DATA_BLOCK "BOTONERA"   // DB2
{ S7_Optimized_Access := 'TRUE' }
VERSION : 0.1
   VAR
      "096P005A" : Struct
         START : Bool;
         STOP : Bool;
         FALLA : Bool;
         "RESET FALLA" : Bool;
         "RESET TIEMPO OPERANDO" : Bool;
         "RESET TIEMPO ACUMULADO" : Bool;
      END_STRUCT;
      "096P005B" : Struct
         START : Bool;
         STOP : Bool;
         FALLA : Bool;
         "RESET FALLA" : Bool;
         "RESET TIEMPO OPERANDO" : Bool;
         "RESET TIEMPO ACUMULADO" : Bool;
      END_STRUCT;
      "096P004A" : Struct
         START : Bool;
         STOP : Bool;
         FALLA : Bool;
         "RESET FALLA" : Bool;
         "RESET TIEMPO OPERANDO" : Bool;
         "RESET TIEMPO ACUMULADO" : Bool;
      END_STRUCT;
      "096P004B" : Struct
         START : Bool;
         STOP : Bool;
         FALLA : Bool;
         "RESET FALLA" : Bool;
         "RESET TIEMPO OPERANDO" : Bool;
         "RESET TIEMPO ACUMULADO" : Bool;
      END_STRUCT;
      "096P004C" : Struct
         START : Bool;
         STOP : Bool;
         FALLA : Bool;
         "RESET FALLA" : Bool;
         "RESET TIEMPO OPERANDO" : Bool;
         "RESET TIEMPO ACUMULADO" : Bool;
      END_STRUCT;
      "096P004D" : Struct
         START : Bool;
         STOP : Bool;
         FALLA : Bool;
         "RESET FALLA" : Bool;
         "RESET TIEMPO OPERANDO" : Bool;
         "RESET TIEMPO ACUMULADO" : Bool;
      END_STRUCT;
      "TODO A MANUAL" : Bool;
      "TODO A AUTOMATICO" : Bool;
      "TODO EN MANUAL" : Bool;
      "TODO EN AUTOMATICO" : Bool;
   END_VAR
BEGIN
END_DATA_BLOCK

DATA_BLOCK "MODO OPERACION"   // DB3
{ S7_Optimized_Access := 'TRUE' }
VERSION : 0.1
   VAR RETAIN
      "096P004A" : Struct
         MANUAL : Bool;
         AUTOMATICO : Bool;
         SCADA : Bool;
      END_STRUCT;
      "096P004B" : Struct
         MANUAL : Bool;
         AUTOMATICO : Bool;
         SCADA : Bool;
      END_STRUCT;
      "096P004C" : Struct
         MANUAL : Bool;
         AUTOMATICO : Bool;
         SCADA : Bool;
      END_STRUCT;
      "096P004D" : Struct
         MANUAL : Bool;
         AUTOMATICO : Bool;
         SCADA : Bool;
      END_STRUCT;
      "096P005A" : Struct
         MANUAL : Bool;
         AUTOMATICO : Bool;
         SCADA : Bool;
      END_STRUCT;
      "096P005B" : Struct
         MANUAL : Bool;
         AUTOMATICO : Bool;
         SCADA : Bool;
      END_STRUCT;
   END_VAR
BEGIN
END_DATA_BLOCK

DATA_BLOCK "ESC HZ"   // DB4
{ S7_Optimized_Access := 'TRUE' }
VERSION : 0.1
   VAR RETAIN
      "096P004A" : Struct
         "FRECUENCIA MAX" : Real := 60.0;
         "FRECUENCIA MIN" : Real := 20.0;
         "FRECUENCIA OP" : Real := 60.0;
      END_STRUCT;
      "096P004B" : Struct
         "FRECUENCIA MAX" : Real := 60.0;
         "FRECUENCIA MIN" : Real := 20.0;
         "FRECUENCIA OP" : Real := 60.0;
      END_STRUCT;
      "096P004C" : Struct
         "FRECUENCIA MAX" : Real := 60.0;
         "FRECUENCIA MIN" : Real := 20.0;
         "FRECUENCIA OP" : Real := 60.0;
      END_STRUCT;
      "096P004D" : Struct
         "FRECUENCIA MAX" : Real := 60.0;
         "FRECUENCIA MIN" : Real := 20.0;
         "FRECUENCIA OP" : Real := 60.0;
      END_STRUCT;
   END_VAR
BEGIN
END_DATA_BLOCK

DATA_BLOCK "DATOS LECTURA VFDS"   // DB5
{ S7_Optimized_Access := 'TRUE' }
VERSION : 0.1
   VAR
      "096P004A" : Struct
         AMPERAJE : Real;
         FRECUENCIA : Real;
         "FRECUENCIA %" : Real;
         VOLTAJE : Real;
         ESTADO : Bool;
      END_STRUCT;
      "096P004B" : Struct
         AMPERAJE : Real;
         FRECUENCIA : Real;
         "FRECUENCIA %" : Real;
         VOLTAJE : Real;
         ESTADO : Bool;
      END_STRUCT;
      "096P004C" : Struct
         AMPERAJE : Real;
         FRECUENCIA : Real;
         "FRECUENCIA %" : Real;
         VOLTAJE : Real;
         ESTADO : Bool;
      END_STRUCT;
      "096P004D" : Struct
         AMPERAJE : Real;
         FRECUENCIA : Real;
         "FRECUENCIA %" : Real;
         VOLTAJE : Real;
         ESTADO : Bool;
      END_STRUCT;
      "096P005A" : Struct
         AMPERAJE : Real;
         FRECUENCIA : Real;
         "FRECUENCIA %" : Real;
         VOLTAJE : Real;
         ESTADO : Bool;
      END_STRUCT;
      "096P005B" : Struct
         AMPERAJE : Real;
         FRECUENCIA : Real;
         "FRECUENCIA %" : Real;
         VOLTAJE : Real;
         ESTADO : Bool;
      END_STRUCT;
   END_VAR
BEGIN
END_DATA_BLOCK

DATA_BLOCK "Alarmas Sis potable y biogas"   // DB6
{ S7_Optimized_Access := 'TRUE' }
VERSION : 0.1
   VAR
      "Alarma general" : Bool;
      "Reset alarmas" : Bool;
   END_VAR
BEGIN
END_DATA_BLOCK

DATA_BLOCK "CONFIG SIS AGUA POTABLE"   // DB25
{ S7_Optimized_Access := 'TRUE' }
VERSION : 0.1
   VAR RETAIN
      "DESVIO DE PRESION PARA DESPERTAR" : Real := 6.0;
      "VALOR DE FRECUENCIA PARA DORMIR" : Real := 34.0;
      "TIEMPO PARA MODO DORMIR" : Real := 40.0;
      "FRECUENCIA PARA ARRANCAR BOMBA EN PARALELO" : Real := 59.0;
      "TIEMPO PARA ARRANCAR BOMBA EN PARALELO" : Real := 10.0;
      "FRECUENCIA PARA APAGAR BOMBA EN PARALELO" : Real := 50.0;
      "TIEMPO PARA APAGAR BOMBA EN PARALELO" : Real := 5.0;
      "TORQUE MINIMO PARA DETECCION BOMBA EN VACIO" : Real := 20.0;
      "TIEMPO DETECCION BOMBA EN VACIO" : Real := 10.0;
      "PRESION BOOSTER" : Real := 2.0;
      "TIEMPO SLEEP BOOSTER" : Real := 10.0;
      "FRECUENCIA MAXIMA CONFIGURADA EN VFDS" : Real := 60.0;
      "FRECUENCIA MINIMA CONFIGURADA EN VFDS" : Real := 33.0;
      "TIEMPO DE ALTERNACION" : Int := 10;
      SETPOINT : Real := 65.0;
      "SETPOINT %" : DInt := 28;
      K : Real := 15.0;
      TI : Real := 20.0;
      TD : Real := 20.0;
   END_VAR
   VAR
      "SALIDA PID %" : Real := 0.0;
   END_VAR
   VAR RETAIN
      "TIEMPO ALTERNACION BOMBAS BIOGAS" : Int := 60;
   END_VAR
BEGIN
END_DATA_BLOCK

DATA_BLOCK "DATOS ESCRITURA VFDS"   // DB30
{ S7_Optimized_Access := 'TRUE' }
VERSION : 0.1
   VAR
      "096P004A" : Struct
         FRECUENCIA : Real;
      END_STRUCT;
      "096P004B" : Struct
         FRECUENCIA : Real;
      END_STRUCT;
      "096P004C" : Struct
         FRECUENCIA : Real;
      END_STRUCT;
      "096P004D" : Struct
         FRECUENCIA : Real;
      END_STRUCT;
   END_VAR
BEGIN
END_DATA_BLOCK

DATA_BLOCK "CP_AS8"   // DB32
{ S7_Optimized_Access := 'TRUE' }
VERSION : 0.1
   VAR
      CONNECT : TCON_IP_v4;
   END_VAR
BEGIN
   CONNECT.InterfaceId := 64;
   CONNECT.ID := 3;
   CONNECT.ConnectionType := 11;
   CONNECT.ActiveEstablished := true;
   CONNECT.RemoteAddress.ADDR[1] := 172;
   CONNECT.RemoteAddress.ADDR[2] := 23;
   CONNECT.RemoteAddress.ADDR[3] := 17;
   CONNECT.RemoteAddress.ADDR[4] := 73;
   CONNECT.RemotePort := 502;
   CONNECT.LocalPort := 504;
END_DATA_BLOCK

DATA_BLOCK "CP_SOFTSTARTER_MODBUS_DB_AS8"   // DB33
{ S7_Optimized_Access := 'FALSE' }
VERSION : 0.1
// stored: InstanceOfName CP_SOFTSTARTER_MODBUS
"CP_SOFTSTARTER_MODBUS"
BEGIN
END_DATA_BLOCK

DATA_BLOCK "DATA MODBUS TCP"   // DB78
{ S7_Optimized_Access := 'FALSE' }
VERSION : 0.1
   VAR
      DATA : Array[0..100] of Word;
   END_VAR
BEGIN
END_DATA_BLOCK

DATA_BLOCK "MB CONFIG"   // DB79
{ S7_Optimized_Access := 'FALSE' }
VERSION : 0.1
   VAR
      CONNECT : TCON_IP_v4;
      NDR : Bool;
      DR : Bool;
      ERROR : Bool;
      STATUS : Word;
   END_VAR
BEGIN
   CONNECT.InterfaceId := 64;
   CONNECT.ID := 1;
   CONNECT.ConnectionType := 11;
   CONNECT.LocalPort := 502;
END_DATA_BLOCK

DATA_BLOCK "CP_SOFTSTARTER_MODBUS_DB_AS7"   // DB80
{ S7_Optimized_Access := 'FALSE' }
VERSION : 0.1
// stored: InstanceOfName CP_SOFTSTARTER_MODBUS
"CP_SOFTSTARTER_MODBUS"
BEGIN
END_DATA_BLOCK

DATA_BLOCK "LECTURA TAB WILO"   // DB91
{ S7_Optimized_Access := 'FALSE' }
VERSION : 0.1
   VAR
      "40014+" : Array[0..6] of Int;
      "40033+" : Array[0..12] of Int;
      "40050+" : Array[0..4] of Int;
   END_VAR
BEGIN
END_DATA_BLOCK

DATA_BLOCK "ESCRITURA TAB WILO"   // DB92
{ S7_Optimized_Access := 'FALSE' }
VERSION : 0.1
   VAR
      "40041+" : Array[0..4] of Int;
      "40016+" : Array[0..4] of Int;
   END_VAR
BEGIN
END_DATA_BLOCK

DATA_BLOCK "FALLAS HMI"   // DB93
{ S7_Optimized_Access := 'FALSE' }
VERSION : 0.1
   VAR
      "PARO EMERGENCIA ACTIVO SISTEMA GRAL AGUA POTABLE Y BIOGAS" : Bool;
      "FALLA GUARDAMOTOR BOMBA 096P005A" : Bool;
      "FALLA GUARDAMOTOR BOMBA 096P005B" : Bool;
      "FALLA ARRANCADOR SUAVE BOMBA P005A" : Bool;
      "FALLA ARRANCADOR SUAVE BOMBA P005B" : Bool;
      "NO CONFIRMA ARRANQUE BOMBA 096P005A" : Bool;
      "PARO DE EMERGENCIA ACTIVO 096P005A" : Bool;
      "NO CONFIRMA ARRANQUE BOMBA 096P005B" : Bool;
      "PARO DE EMERGENCIA ACTIVO 096P005B" : Bool;
      "PARO DE EMERGENCIA ACTIVO 096P004A" : Bool;
      "NO CONFIRMA ARRANQUE BOMBA 096P004A" : Bool;
      "FALLA VARIADOR VELOCIDAD 096P004A" : Bool;
      "PARO DE EMERGENCIA ACTIVO 096P004B" : Bool;
      "NO CONFIRMA ARRANQUE BOMBA 096P004B" : Bool;
      "FALLA VARIADOR VELOCIDAD 096P004B" : Bool;
      "PARO DE EMERGENCIA ACTIVO 096P004C" : Bool;
      "NO CONFIRMA ARRANQUE BOMBA 096P004C" : Bool;
      "FALLA VARIADOR VELOCIDAD 096P004C" : Bool;
      "PARO DE EMERGENCIA ACTIVO 096P004D" : Bool;
      "NO CONFIRMA ARRANQUE BOMBA 096P004D" : Bool;
      "FALLA VARIADOR VELOCIDAD 096P004D" : Bool;
      "SWITCH DE PRESION EN SUCCION INACTIVO PSL005" : Bool;
      "SWITCH DE PRESION EN SUCCION INACTIVO PSL004" : Bool;
      "SWITCH DE PRESION EN SUCCION INACTIVO PSL009" : Bool;
      "NO CONFIRMA SWITCH DE FLUJO CON BOMBA 096P005A" : Bool;
      "NO CONFIRMA SWITCH DE FLUJO CON BOMBA 096P005B" : Bool;
      "NO CONFIRMA SWITCH DE FLUJO CON BOMBA 096P004A" : Bool;
      "NO CONFIRMA SWITCH DE FLUJO CON BOMBA 096P004B" : Bool;
      "NO CONFIRMA SWITCH DE FLUJO CON BOMBA 096P004C" : Bool;
      "NO CONFIRMA SWITCH DE FLUJO CON BOMBA 096P004D" : Bool;
      "FALLA POR ALTA PRESION DE DESCARGA 096PIT008" : Bool;
      "ALARMA POR ALTA PRESION DE DESCARGA 096PIT008" : Bool;
      "ALARMA POR BAJA PRESION DE DESCARGA 096PIT008" : Bool;
      "FALLA POR BAJA PRESION DE DESCARGA 096PIT008" : Bool;
      "FALLA POR ALTA PRESION DE SUCCION 096PIT005" : Bool;
      "ALARMA POR ALTA PRESION DE SUCCION 096PIT005" : Bool;
      "ALARMA POR BAJA PRESION DE SUCCION 096PIT005" : Bool;
      "FALLA POR BAJA PRESION DE SUCCION 096PIT005" : Bool;
      "FALLA POR ALTA PRESION DE DESCARGA 096PIT010" : Bool;
      "ALARMA POR ALTA PRESION DE DESCARGA 096PIT010" : Bool;
      "ALARMA POR BAJA PRESION DE DESCARGA 096PIT010" : Bool;
      "FALLA POR BAJA PRESION DE DESCARGA 096PIT010" : Bool;
      "FALLA POR ALTA PRESION DE SUCCION 096PIT009" : Bool;
      "ALARMA POR ALTA PRESION DE SUCCION 096PIT009" : Bool;
      "ALARMA POR BAJA PRESION DE SUCCION 096PIT009" : Bool;
      "FALLA POR BAJA PRESION DE SUCCION 096PIT009" : Bool;
      "FALLA POR ALTA PRESION DE DESCARGA 096PIT006" : Bool;
      "ALARMA POR ALTA PRESION DE DESCARGA 096PIT006" : Bool;
      "ALARMA POR BAJA PRESION DE DESCARGA 096PIT006" : Bool;
      "FALLA POR BAJA PRESION DE DESCARGA 096PIT006" : Bool;
      "FALLA POR ALTA PRESION DE SUCCION 096PIT004" : Bool;
      "ALARMA POR ALTA PRESION DE SUCCION 096PIT004" : Bool;
      "ALARMA POR BAJA PRESION DE SUCCION 096PIT004" : Bool;
      "FALLA POR BAJA PRESION DE SUCCION 096PIT004" : Bool;
   END_VAR
BEGIN
END_DATA_BLOCK

DATA_BLOCK "CP_AS7"   // DB106
{ S7_Optimized_Access := 'TRUE' }
VERSION : 0.1
   VAR
      CONNECT : TCON_IP_v4;
   END_VAR
BEGIN
   CONNECT.InterfaceId := 64;
   CONNECT.ID := 2;
   CONNECT.ConnectionType := 11;
   CONNECT.ActiveEstablished := true;
   CONNECT.RemoteAddress.ADDR[1] := 172;
   CONNECT.RemoteAddress.ADDR[2] := 23;
   CONNECT.RemoteAddress.ADDR[3] := 17;
   CONNECT.RemoteAddress.ADDR[4] := 72;
   CONNECT.RemotePort := 502;
   CONNECT.LocalPort := 503;
END_DATA_BLOCK

// folder: System blocks/Program resources

DATA_BLOCK "tiempo confirmacion presion 5A"   // DB7
{ S7_Optimized_Access := 'TRUE' }
AUTHOR : Simatic
FAMILY : IEC
NAME : IEC_TMR
VERSION : 1.0
// stored: InstanceOfName IEC_TIMER
"IEC_TIMER"
BEGIN
END_DATA_BLOCK

DATA_BLOCK "tiempo confirmacion presion 5B"   // DB8
{ S7_Optimized_Access := 'TRUE' }
AUTHOR : Simatic
FAMILY : IEC
NAME : IEC_TMR
VERSION : 1.0
// stored: InstanceOfName IEC_TIMER
"IEC_TIMER"
BEGIN
END_DATA_BLOCK

DATA_BLOCK "TEMPO MODO MANUAL 005A"   // DB9
{ S7_Optimized_Access := 'TRUE' }
AUTHOR : Simatic
FAMILY : IEC
NAME : IEC_TMR
VERSION : 1.0
// stored: InstanceOfName IEC_TIMER
"IEC_TIMER"
BEGIN
END_DATA_BLOCK

DATA_BLOCK "TEMPO MODO AUTOMATICO 005A"   // DB10
{ S7_Optimized_Access := 'TRUE' }
AUTHOR : Simatic
FAMILY : IEC
NAME : IEC_TMR
VERSION : 1.0
// stored: InstanceOfName IEC_TIMER
"IEC_TIMER"
BEGIN
END_DATA_BLOCK

DATA_BLOCK "TEMPO MODO SCADA 005A"   // DB11
{ S7_Optimized_Access := 'TRUE' }
AUTHOR : Simatic
FAMILY : IEC
NAME : IEC_TMR
VERSION : 1.0
// stored: InstanceOfName IEC_TIMER
"IEC_TIMER"
BEGIN
END_DATA_BLOCK

DATA_BLOCK "TOF1"   // DB12
{ S7_Optimized_Access := 'TRUE' }
AUTHOR : Simatic
FAMILY : IEC
NAME : IEC_TMR
VERSION : 1.0
// stored: InstanceOfName IEC_TIMER
"IEC_TIMER"
BEGIN
END_DATA_BLOCK

DATA_BLOCK "TEMPO MODO MANUAL 005B"   // DB13
{ S7_Optimized_Access := 'TRUE' }
AUTHOR : Simatic
FAMILY : IEC
NAME : IEC_TMR
VERSION : 1.0
// stored: InstanceOfName IEC_TIMER
"IEC_TIMER"
BEGIN
END_DATA_BLOCK

DATA_BLOCK "TEMPO MODO AUTOMATICO 005B"   // DB14
{ S7_Optimized_Access := 'TRUE' }
AUTHOR : Simatic
FAMILY : IEC
NAME : IEC_TMR
VERSION : 1.0
// stored: InstanceOfName IEC_TIMER
"IEC_TIMER"
BEGIN
END_DATA_BLOCK

DATA_BLOCK "TEMPO MODO SCADA 005B"   // DB15
{ S7_Optimized_Access := 'TRUE' }
AUTHOR : Simatic
FAMILY : IEC
NAME : IEC_TMR
VERSION : 1.0
// stored: InstanceOfName IEC_TIMER
"IEC_TIMER"
BEGIN
END_DATA_BLOCK

DATA_BLOCK "TOF2"   // DB16
{ S7_Optimized_Access := 'TRUE' }
AUTHOR : Simatic
FAMILY : IEC
NAME : IEC_TMR
VERSION : 1.0
// stored: InstanceOfName IEC_TIMER
"IEC_TIMER"
BEGIN
END_DATA_BLOCK

DATA_BLOCK "CONT SEG B5A"   // DB18
{ S7_Optimized_Access := 'TRUE' }
AUTHOR : Simatic
FAMILY : IEC
NAME : CNTR
VERSION : 1.0
// stored: InstanceOfName IEC_COUNTER
"IEC_COUNTER"
BEGIN
END_DATA_BLOCK

DATA_BLOCK "CONT MIN B5A"   // DB19
{ S7_Optimized_Access := 'TRUE' }
AUTHOR : Simatic
FAMILY : IEC
NAME : CNTR
VERSION : 1.0
// stored: InstanceOfName IEC_COUNTER
"IEC_COUNTER"
BEGIN
END_DATA_BLOCK

DATA_BLOCK "RESET B5A"   // DB20
{ S7_Optimized_Access := 'TRUE' }
AUTHOR : Simatic
FAMILY : IEC
NAME : IEC_TMR
VERSION : 1.0
// stored: InstanceOfName IEC_TIMER
"IEC_TIMER"
BEGIN
END_DATA_BLOCK

DATA_BLOCK "CONT SEG B5B"   // DB21
{ S7_Optimized_Access := 'TRUE' }
AUTHOR : Simatic
FAMILY : IEC
NAME : CNTR
VERSION : 1.0
// stored: InstanceOfName IEC_COUNTER
"IEC_COUNTER"
BEGIN
END_DATA_BLOCK

DATA_BLOCK "CONT MIN B5B"   // DB22
{ S7_Optimized_Access := 'TRUE' }
AUTHOR : Simatic
FAMILY : IEC
NAME : CNTR
VERSION : 1.0
// stored: InstanceOfName IEC_COUNTER
"IEC_COUNTER"
BEGIN
END_DATA_BLOCK

DATA_BLOCK "RESET B5B"   // DB23
{ S7_Optimized_Access := 'TRUE' }
AUTHOR : Simatic
FAMILY : IEC
NAME : IEC_TMR
VERSION : 1.0
// stored: InstanceOfName IEC_TIMER
"IEC_TIMER"
BEGIN
END_DATA_BLOCK

DATA_BLOCK "CONTADOR ALTERNACION BIOGAS"   // DB24
{ S7_Optimized_Access := 'TRUE' }
AUTHOR : Simatic
FAMILY : IEC
NAME : CNTR
VERSION : 1.0
// stored: InstanceOfName IEC_COUNTER
"IEC_COUNTER"
BEGIN
END_DATA_BLOCK

DATA_BLOCK "FALLA BOMBA LIDER BIOGAS 1"   // DB26
{ S7_Optimized_Access := 'TRUE' }
AUTHOR : Simatic
FAMILY : IEC
NAME : IEC_TMR
VERSION : 1.0
// stored: InstanceOfName IEC_TIMER
"IEC_TIMER"
BEGIN
END_DATA_BLOCK

DATA_BLOCK "FALLA BOMBA LIDER BIOGAS 2"   // DB27
{ S7_Optimized_Access := 'TRUE' }
AUTHOR : Simatic
FAMILY : IEC
NAME : IEC_TMR
VERSION : 1.0
// stored: InstanceOfName IEC_TIMER
"IEC_TIMER"
BEGIN
END_DATA_BLOCK

DATA_BLOCK "tiempo confirmacion presion 4"   // DB28
{ S7_Optimized_Access := 'TRUE' }
AUTHOR : Simatic
FAMILY : IEC
NAME : IEC_TMR
VERSION : 1.0
// stored: InstanceOfName IEC_TIMER
"IEC_TIMER"
BEGIN
END_DATA_BLOCK

DATA_BLOCK "TEMPO MODO MANUAL 004A"   // DB29
{ S7_Optimized_Access := 'TRUE' }
AUTHOR : Simatic
FAMILY : IEC
NAME : IEC_TMR
VERSION : 1.0
// stored: InstanceOfName IEC_TIMER
"IEC_TIMER"
BEGIN
END_DATA_BLOCK

DATA_BLOCK "TEMPO MODO SCADA 004A"   // DB31
{ S7_Optimized_Access := 'TRUE' }
AUTHOR : Simatic
FAMILY : IEC
NAME : IEC_TMR
VERSION : 1.0
// stored: InstanceOfName IEC_TIMER
"IEC_TIMER"
BEGIN
END_DATA_BLOCK

DATA_BLOCK "TOF11"   // DB34
{ S7_Optimized_Access := 'TRUE' }
AUTHOR : Simatic
FAMILY : IEC
NAME : IEC_TMR
VERSION : 1.0
// stored: InstanceOfName IEC_TIMER
"IEC_TIMER"
BEGIN
END_DATA_BLOCK

DATA_BLOCK "TEMPO MODO MANUAL 004B"   // DB35
{ S7_Optimized_Access := 'TRUE' }
AUTHOR : Simatic
FAMILY : IEC
NAME : IEC_TMR
VERSION : 1.0
// stored: InstanceOfName IEC_TIMER
"IEC_TIMER"
BEGIN
END_DATA_BLOCK

DATA_BLOCK "TEMPO MODO AUTOMATICO 004B"   // DB36
{ S7_Optimized_Access := 'TRUE' }
AUTHOR : Simatic
FAMILY : IEC
NAME : IEC_TMR
VERSION : 1.0
// stored: InstanceOfName IEC_TIMER
"IEC_TIMER"
BEGIN
END_DATA_BLOCK

DATA_BLOCK "TEMPO MODO SCADA 004B"   // DB37
{ S7_Optimized_Access := 'TRUE' }
AUTHOR : Simatic
FAMILY : IEC
NAME : IEC_TMR
VERSION : 1.0
// stored: InstanceOfName IEC_TIMER
"IEC_TIMER"
BEGIN
END_DATA_BLOCK

DATA_BLOCK "TOF12"   // DB38
{ S7_Optimized_Access := 'TRUE' }
AUTHOR : Simatic
FAMILY : IEC
NAME : IEC_TMR
VERSION : 1.0
// stored: InstanceOfName IEC_TIMER
"IEC_TIMER"
BEGIN
END_DATA_BLOCK

DATA_BLOCK "TEMPO MODO MANUAL 004C"   // DB39
{ S7_Optimized_Access := 'TRUE' }
AUTHOR : Simatic
FAMILY : IEC
NAME : IEC_TMR
VERSION : 1.0
// stored: InstanceOfName IEC_TIMER
"IEC_TIMER"
BEGIN
END_DATA_BLOCK

DATA_BLOCK "TEMPO MODO AUTOMATICO 004C"   // DB40
{ S7_Optimized_Access := 'TRUE' }
AUTHOR : Simatic
FAMILY : IEC
NAME : IEC_TMR
VERSION : 1.0
// stored: InstanceOfName IEC_TIMER
"IEC_TIMER"
BEGIN
END_DATA_BLOCK

DATA_BLOCK "TEMPO MODO SCADA 004C"   // DB41
{ S7_Optimized_Access := 'TRUE' }
AUTHOR : Simatic
FAMILY : IEC
NAME : IEC_TMR
VERSION : 1.0
// stored: InstanceOfName IEC_TIMER
"IEC_TIMER"
BEGIN
END_DATA_BLOCK

DATA_BLOCK "TOF13"   // DB42
{ S7_Optimized_Access := 'TRUE' }
AUTHOR : Simatic
FAMILY : IEC
NAME : IEC_TMR
VERSION : 1.0
// stored: InstanceOfName IEC_TIMER
"IEC_TIMER"
BEGIN
END_DATA_BLOCK

DATA_BLOCK "TEMPO MODO MANUAL 004D"   // DB43
{ S7_Optimized_Access := 'TRUE' }
AUTHOR : Simatic
FAMILY : IEC
NAME : IEC_TMR
VERSION : 1.0
// stored: InstanceOfName IEC_TIMER
"IEC_TIMER"
BEGIN
END_DATA_BLOCK

DATA_BLOCK "TEMPO MODO AUTOMATICO 004D"   // DB44
{ S7_Optimized_Access := 'TRUE' }
AUTHOR : Simatic
FAMILY : IEC
NAME : IEC_TMR
VERSION : 1.0
// stored: InstanceOfName IEC_TIMER
"IEC_TIMER"
BEGIN
END_DATA_BLOCK

DATA_BLOCK "TEMPO MODO SCADA 004D"   // DB45
{ S7_Optimized_Access := 'TRUE' }
AUTHOR : Simatic
FAMILY : IEC
NAME : IEC_TMR
VERSION : 1.0
// stored: InstanceOfName IEC_TIMER
"IEC_TIMER"
BEGIN
END_DATA_BLOCK

DATA_BLOCK "TOF14"   // DB46
{ S7_Optimized_Access := 'TRUE' }
AUTHOR : Simatic
FAMILY : IEC
NAME : IEC_TMR
VERSION : 1.0
// stored: InstanceOfName IEC_TIMER
"IEC_TIMER"
BEGIN
END_DATA_BLOCK

DATA_BLOCK "PRES OK"   // DB48
{ S7_Optimized_Access := 'TRUE' }
AUTHOR : Simatic
FAMILY : IEC
NAME : IEC_TMR
VERSION : 1.0
// stored: InstanceOfName IEC_TIMER
"IEC_TIMER"
BEGIN
END_DATA_BLOCK

DATA_BLOCK "TIEMPO PARA APAGAR"   // DB49
{ S7_Optimized_Access := 'TRUE' }
AUTHOR : Simatic
FAMILY : IEC
NAME : IEC_TMR
VERSION : 1.0
// stored: InstanceOfName IEC_TIMER
"IEC_TIMER"
BEGIN
END_DATA_BLOCK

DATA_BLOCK "TIEMPO SLEEP BOOSTER"   // DB50
{ S7_Optimized_Access := 'TRUE' }
AUTHOR : Simatic
FAMILY : IEC
NAME : IEC_TMR
VERSION : 1.0
// stored: InstanceOfName IEC_TIMER
"IEC_TIMER"
BEGIN
END_DATA_BLOCK

DATA_BLOCK "RESET SLEEP BOOSTER"   // DB51
{ S7_Optimized_Access := 'TRUE' }
AUTHOR : Simatic
FAMILY : IEC
NAME : IEC_TMR
VERSION : 1.0
// stored: InstanceOfName IEC_TIMER
"IEC_TIMER"
BEGIN
END_DATA_BLOCK

DATA_BLOCK "CONT SEG BA"   // DB52
{ S7_Optimized_Access := 'TRUE' }
AUTHOR : Simatic
FAMILY : IEC
NAME : CNTR
VERSION : 1.0
// stored: InstanceOfName IEC_COUNTER
"IEC_COUNTER"
BEGIN
END_DATA_BLOCK

DATA_BLOCK "CONT MIN BA"   // DB53
{ S7_Optimized_Access := 'TRUE' }
AUTHOR : Simatic
FAMILY : IEC
NAME : CNTR
VERSION : 1.0
// stored: InstanceOfName IEC_COUNTER
"IEC_COUNTER"
BEGIN
END_DATA_BLOCK

DATA_BLOCK "RESET BA"   // DB54
{ S7_Optimized_Access := 'TRUE' }
AUTHOR : Simatic
FAMILY : IEC
NAME : IEC_TMR
VERSION : 1.0
// stored: InstanceOfName IEC_TIMER
"IEC_TIMER"
BEGIN
END_DATA_BLOCK

DATA_BLOCK "CONT SEG BB"   // DB55
{ S7_Optimized_Access := 'TRUE' }
AUTHOR : Simatic
FAMILY : IEC
NAME : CNTR
VERSION : 1.0
// stored: InstanceOfName IEC_COUNTER
"IEC_COUNTER"
BEGIN
END_DATA_BLOCK

DATA_BLOCK "CONT MIN BB"   // DB56
{ S7_Optimized_Access := 'TRUE' }
AUTHOR : Simatic
FAMILY : IEC
NAME : CNTR
VERSION : 1.0
// stored: InstanceOfName IEC_COUNTER
"IEC_COUNTER"
BEGIN
END_DATA_BLOCK

DATA_BLOCK "RESET BB"   // DB57
{ S7_Optimized_Access := 'TRUE' }
AUTHOR : Simatic
FAMILY : IEC
NAME : IEC_TMR
VERSION : 1.0
// stored: InstanceOfName IEC_TIMER
"IEC_TIMER"
BEGIN
END_DATA_BLOCK

DATA_BLOCK "CONT SEG BC"   // DB58
{ S7_Optimized_Access := 'TRUE' }
AUTHOR : Simatic
FAMILY : IEC
NAME : CNTR
VERSION : 1.0
// stored: InstanceOfName IEC_COUNTER
"IEC_COUNTER"
BEGIN
END_DATA_BLOCK

DATA_BLOCK "CONT MIN BC"   // DB59
{ S7_Optimized_Access := 'TRUE' }
AUTHOR : Simatic
FAMILY : IEC
NAME : CNTR
VERSION : 1.0
// stored: InstanceOfName IEC_COUNTER
"IEC_COUNTER"
BEGIN
END_DATA_BLOCK

DATA_BLOCK "RESET BC"   // DB60
{ S7_Optimized_Access := 'TRUE' }
AUTHOR : Simatic
FAMILY : IEC
NAME : IEC_TMR
VERSION : 1.0
// stored: InstanceOfName IEC_TIMER
"IEC_TIMER"
BEGIN
END_DATA_BLOCK

DATA_BLOCK "CONT SEG BD"   // DB61
{ S7_Optimized_Access := 'TRUE' }
AUTHOR : Simatic
FAMILY : IEC
NAME : CNTR
VERSION : 1.0
// stored: InstanceOfName IEC_COUNTER
"IEC_COUNTER"
BEGIN
END_DATA_BLOCK

DATA_BLOCK "CONT MIN BD"   // DB62
{ S7_Optimized_Access := 'TRUE' }
AUTHOR : Simatic
FAMILY : IEC
NAME : CNTR
VERSION : 1.0
// stored: InstanceOfName IEC_COUNTER
"IEC_COUNTER"
BEGIN
END_DATA_BLOCK

DATA_BLOCK "RESET BD"   // DB63
{ S7_Optimized_Access := 'TRUE' }
AUTHOR : Simatic
FAMILY : IEC
NAME : IEC_TMR
VERSION : 1.0
// stored: InstanceOfName IEC_TIMER
"IEC_TIMER"
BEGIN
END_DATA_BLOCK

DATA_BLOCK "CONTADOR ALTERNACION 1"   // DB64
{ S7_Optimized_Access := 'TRUE' }
AUTHOR : Simatic
FAMILY : IEC
NAME : CNTR
VERSION : 1.0
// stored: InstanceOfName IEC_COUNTER
"IEC_COUNTER"
BEGIN
END_DATA_BLOCK

DATA_BLOCK "FALLA BOMBA LIDER 1"   // DB65
{ S7_Optimized_Access := 'TRUE' }
AUTHOR : Simatic
FAMILY : IEC
NAME : IEC_TMR
VERSION : 1.0
// stored: InstanceOfName IEC_TIMER
"IEC_TIMER"
BEGIN
END_DATA_BLOCK

DATA_BLOCK "FALLA BOMBA LIDER 2"   // DB66
{ S7_Optimized_Access := 'TRUE' }
AUTHOR : Simatic
FAMILY : IEC
NAME : IEC_TMR
VERSION : 1.0
// stored: InstanceOfName IEC_TIMER
"IEC_TIMER"
BEGIN
END_DATA_BLOCK

DATA_BLOCK "FALLA BOMBA LIDER 3"   // DB67
{ S7_Optimized_Access := 'TRUE' }
AUTHOR : Simatic
FAMILY : IEC
NAME : IEC_TMR
VERSION : 1.0
// stored: InstanceOfName IEC_TIMER
"IEC_TIMER"
BEGIN
END_DATA_BLOCK

DATA_BLOCK "FALLA BOMBA LIDER 4"   // DB68
{ S7_Optimized_Access := 'TRUE' }
AUTHOR : Simatic
FAMILY : IEC
NAME : IEC_TMR
VERSION : 1.0
// stored: InstanceOfName IEC_TIMER
"IEC_TIMER"
BEGIN
END_DATA_BLOCK

DATA_BLOCK "TIEMPO AD1"   // DB69
{ S7_Optimized_Access := 'TRUE' }
AUTHOR : Simatic
FAMILY : IEC
NAME : IEC_TMR
VERSION : 1.0
// stored: InstanceOfName IEC_TIMER
"IEC_TIMER"
BEGIN
END_DATA_BLOCK

DATA_BLOCK "TIEMPO AD2"   // DB70
{ S7_Optimized_Access := 'TRUE' }
AUTHOR : Simatic
FAMILY : IEC
NAME : IEC_TMR
VERSION : 1.0
// stored: InstanceOfName IEC_TIMER
"IEC_TIMER"
BEGIN
END_DATA_BLOCK

DATA_BLOCK "TIEMPO AD3"   // DB71
{ S7_Optimized_Access := 'TRUE' }
AUTHOR : Simatic
FAMILY : IEC
NAME : IEC_TMR
VERSION : 1.0
// stored: InstanceOfName IEC_TIMER
"IEC_TIMER"
BEGIN
END_DATA_BLOCK

DATA_BLOCK "CONT MIN BOMBA A ACUM"   // DB72
{ S7_Optimized_Access := 'TRUE' }
AUTHOR : Simatic
FAMILY : IEC
NAME : CNTR
VERSION : 1.0
// stored: InstanceOfName IEC_COUNTER
"IEC_COUNTER"
BEGIN
END_DATA_BLOCK

DATA_BLOCK "CONT H BOMBA A ACUM"   // DB73
{ S7_Optimized_Access := 'TRUE' }
AUTHOR : Simatic
FAMILY : IEC
NAME : CNTR
VERSION : 1.0
// stored: InstanceOfName IEC_COUNTER
"IEC_COUNTER"
BEGIN
END_DATA_BLOCK

DATA_BLOCK "CONT MIN BOMBA B ACUM"   // DB74
{ S7_Optimized_Access := 'TRUE' }
AUTHOR : Simatic
FAMILY : IEC
NAME : CNTR
VERSION : 1.0
// stored: InstanceOfName IEC_COUNTER
"IEC_COUNTER"
BEGIN
END_DATA_BLOCK

DATA_BLOCK "CONT H BOMBA B ACUM"   // DB75
{ S7_Optimized_Access := 'TRUE' }
AUTHOR : Simatic
FAMILY : IEC
NAME : CNTR
VERSION : 1.0
// stored: InstanceOfName IEC_COUNTER
"IEC_COUNTER"
BEGIN
END_DATA_BLOCK

DATA_BLOCK "CONT MIN BOMBA C ACUM"   // DB76
{ S7_Optimized_Access := 'TRUE' }
AUTHOR : Simatic
FAMILY : IEC
NAME : CNTR
VERSION : 1.0
// stored: InstanceOfName IEC_COUNTER
"IEC_COUNTER"
BEGIN
END_DATA_BLOCK

DATA_BLOCK "CONT H BOMBA C ACUM"   // DB77
{ S7_Optimized_Access := 'TRUE' }
AUTHOR : Simatic
FAMILY : IEC
NAME : CNTR
VERSION : 1.0
// stored: InstanceOfName IEC_COUNTER
"IEC_COUNTER"
BEGIN
END_DATA_BLOCK

DATA_BLOCK "CONT MIN BOMBA D ACUM"   // DB81
{ S7_Optimized_Access := 'TRUE' }
AUTHOR : Simatic
FAMILY : IEC
NAME : CNTR
VERSION : 1.0
// stored: InstanceOfName IEC_COUNTER
"IEC_COUNTER"
BEGIN
END_DATA_BLOCK

DATA_BLOCK "CONT H BOMBA D ACUM"   // DB82
{ S7_Optimized_Access := 'TRUE' }
AUTHOR : Simatic
FAMILY : IEC
NAME : CNTR
VERSION : 1.0
// stored: InstanceOfName IEC_COUNTER
"IEC_COUNTER"
BEGIN
END_DATA_BLOCK

DATA_BLOCK "CONT MIN BOMBA 5A ACUM"   // DB83
{ S7_Optimized_Access := 'TRUE' }
AUTHOR : Simatic
FAMILY : IEC
NAME : CNTR
VERSION : 1.0
// stored: InstanceOfName IEC_COUNTER
"IEC_COUNTER"
BEGIN
END_DATA_BLOCK

DATA_BLOCK "CONT H BOMBA 5A ACUM"   // DB84
{ S7_Optimized_Access := 'TRUE' }
AUTHOR : Simatic
FAMILY : IEC
NAME : CNTR
VERSION : 1.0
// stored: InstanceOfName IEC_COUNTER
"IEC_COUNTER"
BEGIN
END_DATA_BLOCK

DATA_BLOCK "CONT MIN BOMBA 5B ACUM"   // DB85
{ S7_Optimized_Access := 'TRUE' }
AUTHOR : Simatic
FAMILY : IEC
NAME : CNTR
VERSION : 1.0
// stored: InstanceOfName IEC_COUNTER
"IEC_COUNTER"
BEGIN
END_DATA_BLOCK

DATA_BLOCK "CONT H BOMBA 5B ACUM"   // DB86
{ S7_Optimized_Access := 'TRUE' }
AUTHOR : Simatic
FAMILY : IEC
NAME : CNTR
VERSION : 1.0
// stored: InstanceOfName IEC_COUNTER
"IEC_COUNTER"
BEGIN
END_DATA_BLOCK

DATA_BLOCK "TEMPO MODO AUTOMATICO 004A"   // DB87
{ S7_Optimized_Access := 'TRUE' }
AUTHOR : Simatic
FAMILY : IEC
NAME : IEC_TMR
VERSION : 1.0
// stored: InstanceOfName IEC_TIMER
"IEC_TIMER"
BEGIN
END_DATA_BLOCK

DATA_BLOCK "CONTADOR COMUNICACION"   // DB88
{ S7_Optimized_Access := 'TRUE' }
AUTHOR : Simatic
FAMILY : IEC
NAME : CNTR
VERSION : 1.0
// stored: InstanceOfName IEC_COUNTER
"IEC_COUNTER"
BEGIN
END_DATA_BLOCK

DATA_BLOCK "TIEMPO CONFIRMACION 096P004A"   // DB89
{ S7_Optimized_Access := 'TRUE' }
AUTHOR : Simatic
FAMILY : IEC
NAME : IEC_TMR
VERSION : 1.0
// stored: InstanceOfName IEC_TIMER
"IEC_TIMER"
BEGIN
END_DATA_BLOCK

DATA_BLOCK "CONFIRMACION FLUJO 096P004a"   // DB94
{ S7_Optimized_Access := 'TRUE' }
AUTHOR : Simatic
FAMILY : IEC
NAME : IEC_TMR
VERSION : 1.0
// stored: InstanceOfName IEC_TIMER
"IEC_TIMER"
BEGIN
END_DATA_BLOCK

DATA_BLOCK "TIEMPO CONFIRMACION 096P004B"   // DB95
{ S7_Optimized_Access := 'TRUE' }
AUTHOR : Simatic
FAMILY : IEC
NAME : IEC_TMR
VERSION : 1.0
// stored: InstanceOfName IEC_TIMER
"IEC_TIMER"
BEGIN
END_DATA_BLOCK

DATA_BLOCK "CONFIRMACION FLUJO 096P004B"   // DB96
{ S7_Optimized_Access := 'TRUE' }
AUTHOR : Simatic
FAMILY : IEC
NAME : IEC_TMR
VERSION : 1.0
// stored: InstanceOfName IEC_TIMER
"IEC_TIMER"
BEGIN
END_DATA_BLOCK

DATA_BLOCK "TIEMPO CONFIRMACION 096P004C"   // DB97
{ S7_Optimized_Access := 'TRUE' }
AUTHOR : Simatic
FAMILY : IEC
NAME : IEC_TMR
VERSION : 1.0
// stored: InstanceOfName IEC_TIMER
"IEC_TIMER"
BEGIN
END_DATA_BLOCK

DATA_BLOCK "CONFIRMACION FLUJO 096P004C"   // DB98
{ S7_Optimized_Access := 'TRUE' }
AUTHOR : Simatic
FAMILY : IEC
NAME : IEC_TMR
VERSION : 1.0
// stored: InstanceOfName IEC_TIMER
"IEC_TIMER"
BEGIN
END_DATA_BLOCK

DATA_BLOCK "TIEMPO CONFIRMACION 096P004D"   // DB100
{ S7_Optimized_Access := 'TRUE' }
AUTHOR : Simatic
FAMILY : IEC
NAME : IEC_TMR
VERSION : 1.0
// stored: InstanceOfName IEC_TIMER
"IEC_TIMER"
BEGIN
END_DATA_BLOCK

DATA_BLOCK "CONFIRMACION FLUJO 096P004D"   // DB101
{ S7_Optimized_Access := 'TRUE' }
AUTHOR : Simatic
FAMILY : IEC
NAME : IEC_TMR
VERSION : 1.0
// stored: InstanceOfName IEC_TIMER
"IEC_TIMER"
BEGIN
END_DATA_BLOCK

DATA_BLOCK "TIEMPO CONFIRMACION 096P005A"   // DB102
{ S7_Optimized_Access := 'TRUE' }
AUTHOR : Simatic
FAMILY : IEC
NAME : IEC_TMR
VERSION : 1.0
// stored: InstanceOfName IEC_TIMER
"IEC_TIMER"
BEGIN
END_DATA_BLOCK

DATA_BLOCK "CONFIRMACION FLUJO 096P005A"   // DB103
{ S7_Optimized_Access := 'TRUE' }
AUTHOR : Simatic
FAMILY : IEC
NAME : IEC_TMR
VERSION : 1.0
// stored: InstanceOfName IEC_TIMER
"IEC_TIMER"
BEGIN
END_DATA_BLOCK

DATA_BLOCK "TIEMPO CONFIRMACION 096P005B"   // DB104
{ S7_Optimized_Access := 'TRUE' }
AUTHOR : Simatic
FAMILY : IEC
NAME : IEC_TMR
VERSION : 1.0
// stored: InstanceOfName IEC_TIMER
"IEC_TIMER"
BEGIN
END_DATA_BLOCK

DATA_BLOCK "CONFIRMACION FLUJO 096P005B"   // DB105
{ S7_Optimized_Access := 'TRUE' }
AUTHOR : Simatic
FAMILY : IEC
NAME : IEC_TMR
VERSION : 1.0
// stored: InstanceOfName IEC_TIMER
"IEC_TIMER"
BEGIN
END_DATA_BLOCK

// folder: (top level)

FUNCTION_BLOCK "CP_SOFTSTARTER_MODBUS"   // FB3, SCL
{ S7_Optimized_Access := 'FALSE' }
VERSION : 0.1
   VAR_INPUT
      I_CMD_ON : Bool;
   END_VAR
   VAR_OUTPUT
      O_COMM_ERROR : Bool;
      O_Ready : Bool;
      O_NoMainPower : Bool;
      O_MotorON : Bool;
      O_MotorOverload : Bool;
      O_Fault : Bool;
      O_CurrentLimitExceeded : Bool;
      O_CurrentLimitUndershot : Bool;
      O_AutomaticMode : Bool;
      O_ManualBus : Bool;
      O_ManualLocal : Bool;
      O_PhaseFailureL1 : Bool;
      O_PhaseFailureL2 : Bool;
      O_PhaseFailureL3 : Bool;
      O_BypassDefective : Bool;
      O_CurrentAVG : Real;
   END_VAR
   VAR_IN_OUT
      IO_WP_CONNECT : Variant;
   END_VAR
   VAR
      S_MB_CLIENT_WP : MB_CLIENT;
      S_COMM_PARAMETERS : Struct
         REQ : Bool;
         DISCONNECT : Bool;
         MB_MODE : USInt;
         MB_DATA_ADDR : UDInt;
         MB_DATA_LEN : UInt;
      END_STRUCT;
      S_DATA_PTR : Array[0..999] of Byte;
      S_DATA : Struct
         "BIT_STATUS 1" : Word;
         "BIT_STATUS 2" : Word;
         GROSS_W : DWord;
         NET_W : DWord;
         TARE_W : DWord;
         G_OR_N : DWord;
         D_IN : Word;
      END_STRUCT;
      S_STEP_COMM : Int := 1;
      S_DataSetProcessImageInput : "typeProcessImageInput";
      S_DataSetSoftStarterDiagnostics : "typeSoftStarterDiagnostics";
      S_DataSetMeasuredValues : "typeMeasuredValues";
      S_DataSetProcessImageOutput : "typeProcessImageOutput";
      S_Current : DInt;
   END_VAR
   VAR_TEMP
      T_NOT_CMD : Bool;
      tempPOS : DInt;
      tempRetVal : Int;
      tempPOS_ser : DInt;
      tempRetVal_ser : Int;
   END_VAR
BEGIN
   REGION MB_CLIENT
       // Statement section REGION
       // 
       #S_MB_CLIENT_WP(REQ := #S_COMM_PARAMETERS.REQ,
                       DISCONNECT := #S_COMM_PARAMETERS.DISCONNECT,
                       MB_MODE := #S_COMM_PARAMETERS.#MB_MODE,
                       MB_DATA_ADDR := #S_COMM_PARAMETERS.#MB_DATA_ADDR,
                       MB_DATA_LEN := #S_COMM_PARAMETERS.#MB_DATA_LEN,
                       MB_DATA_PTR := #S_DATA_PTR,
                       CONNECT := #IO_WP_CONNECT);

   END_REGION

   REGION COMM ERROR
       // Statement section REGION
       IF #S_MB_CLIENT_WP.Connected = TRUE THEN
           // Statement section IF
           // 
           #O_COMM_ERROR := FALSE;
       ELSE
           #O_COMM_ERROR := TRUE;
           ;
       END_IF;

   END_REGION

   CASE #S_STEP_COMM OF

       1:  // Read process image input
           REGION READ PROCESS IMAGE INPUT

               #S_COMM_PARAMETERS.#MB_MODE := 103;
               #S_COMM_PARAMETERS.#MB_DATA_ADDR := 32768;
               #S_COMM_PARAMETERS.#MB_DATA_LEN := 8;

               #S_COMM_PARAMETERS.#REQ := NOT #S_MB_CLIENT_WP.BUSY;

               IF #S_MB_CLIENT_WP.DONE THEN
                   // Statement section IF
                   // 
                   #tempRetVal := Deserialize(SRC_ARRAY := #S_DATA_PTR, DEST_VARIABLE => #S_DataSetProcessImageInput, POS := #tempPOS);

                   #S_COMM_PARAMETERS.#REQ := FALSE;
                   #S_STEP_COMM := 2;
                   ;
               END_IF;
           END_REGION
           ;

       2:  // Read diagnostics
           REGION READ DIAGNOSTICS

               #S_COMM_PARAMETERS.#MB_MODE := 103;
               #S_COMM_PARAMETERS.#MB_DATA_ADDR := 33792;
               #S_COMM_PARAMETERS.#MB_DATA_LEN := 42;

               #S_COMM_PARAMETERS.#REQ := NOT #S_MB_CLIENT_WP.BUSY;

               IF #S_MB_CLIENT_WP.DONE THEN
                   // Statement section IF
                   // 
                   #tempRetVal := Deserialize(SRC_ARRAY := #S_DATA_PTR, DEST_VARIABLE => #S_DataSetSoftStarterDiagnostics, POS := #tempPOS);

                   #S_COMM_PARAMETERS.#REQ := FALSE;
                   #S_STEP_COMM := 3;
                   ;
               END_IF;
           END_REGION
           ;
       3:  // Read measured values
           REGION READ MEASURED VALUES

               // #S_COMM_PARAMETERS.#MB_MODE := 103;
               // #S_COMM_PARAMETERS.#MB_DATA_ADDR := 34816;
               // #S_COMM_PARAMETERS.#MB_DATA_LEN := 45;
               // 

               #S_COMM_PARAMETERS.#MB_MODE := 103;
               #S_COMM_PARAMETERS.#MB_DATA_ADDR := 34851;
               #S_COMM_PARAMETERS.#MB_DATA_LEN := 2;

               #S_COMM_PARAMETERS.#REQ := NOT #S_MB_CLIENT_WP.BUSY;

               IF #S_MB_CLIENT_WP.DONE THEN
                   // Statement section IF

                   //#tempRetVal := Deserialize(SRC_ARRAY := #S_DATA_PTR, DEST_VARIABLE => #CP_dataSetMeasuredValues, POS := #tempPOS);

                   #S_Current.%B3 := #S_DATA_PTR[0];
                   #S_Current.%B2 := #S_DATA_PTR[1];
                   #S_Current.%B1 := #S_DATA_PTR[2];
                   #S_Current.%B0 := #S_DATA_PTR[3];

                   #S_COMM_PARAMETERS.#REQ := FALSE;
                   #S_STEP_COMM := 4;
                   ;
               END_IF;

           END_REGION
           ;
       4:  // Write image output
           REGION WRITE IMAGE OUTPUT

               #S_COMM_PARAMETERS.#MB_MODE := 116;
               #S_COMM_PARAMETERS.#MB_DATA_ADDR := 33280;
               #S_COMM_PARAMETERS.#MB_DATA_LEN := 2;

               #S_DataSetProcessImageOutput.motorRight := #I_CMD_ON;
               #tempRetVal_ser := Serialize(SRC_VARIABLE := #S_DataSetProcessImageOutput, DEST_ARRAY => #S_DATA_PTR, POS := #tempPOS_ser);

               #S_COMM_PARAMETERS.#REQ := NOT #S_MB_CLIENT_WP.BUSY;

               IF #S_MB_CLIENT_WP.DONE THEN
                   // Statement section IF
                   // 

                   #S_COMM_PARAMETERS.#REQ := FALSE;
                   #S_STEP_COMM := 1;
                   ;
               END_IF;


           END_REGION
           ;
       ELSE  // Statement section ELSE

           #S_STEP_COMM := 1;
           ;
   END_CASE;

   REGION PROCCESS VALUES OUTPUT
       // Statement section REGION
       // 
       #O_Ready := #S_DataSetSoftStarterDiagnostics.readyToStartForMotorOn;
       #O_NoMainPower := #S_DataSetSoftStarterDiagnostics.noMainPower;
       #O_MotorON := #S_DataSetProcessImageInput.motorOn;
       #O_MotorOverload := #S_DataSetSoftStarterDiagnostics.mototrOverloadShutoff;
       #O_Fault := #S_DataSetSoftStarterDiagnostics.groupError;
       #O_CurrentLimitExceeded := #S_DataSetSoftStarterDiagnostics.currentLimitErrorExceeded;
       #O_CurrentLimitUndershot := #S_DataSetSoftStarterDiagnostics.currentLimitErrorUndershot;
       #O_AutomaticMode := #S_DataSetSoftStarterDiagnostics.automaticMode;
       #O_ManualBus := #S_DataSetSoftStarterDiagnostics.operatingModeManual;
       #O_ManualLocal := #S_DataSetSoftStarterDiagnostics.manualOperationLocal;
       #O_PhaseFailureL1 := #S_DataSetSoftStarterDiagnostics.phaseFailureL1;
       #O_PhaseFailureL2 := #S_DataSetSoftStarterDiagnostics.phaseFailureL2;
       #O_PhaseFailureL3 := #S_DataSetSoftStarterDiagnostics.phaseFailureL3;
       #O_BypassDefective := #S_DataSetSoftStarterDiagnostics.bypassDefective;
       #O_CurrentAVG := DINT_TO_REAL(#S_Current)/100.0;

   END_REGION
END_FUNCTION_BLOCK

FUNCTION "Escalizacion analogas" : Void   // FC1, LAD
{ S7_Optimized_Access := 'TRUE' }
VERSION : 0.1
BEGIN

REGION Network 1: 096PIT005
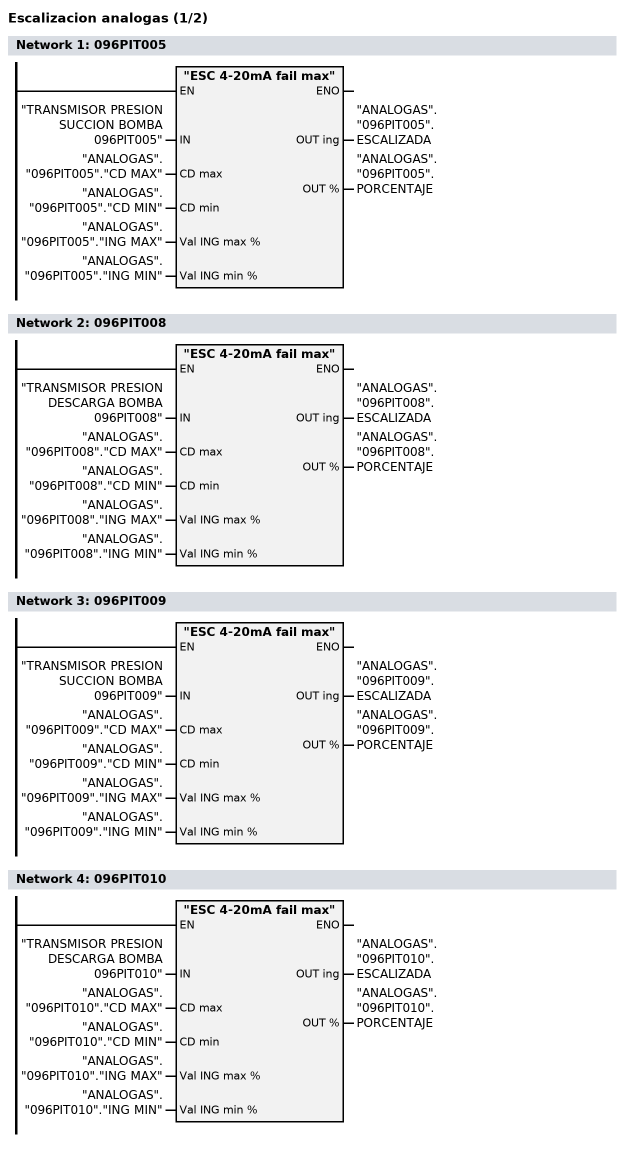
   RUNG wire#powerrail
      "ESC 4-20mA fail max"(IN := "TRANSMISOR PRESION SUCCION BOMBA 096PIT005", "CD max" := "ANALOGAS"."096PIT005"."CD MAX", "CD min" := "ANALOGAS"."096PIT005"."CD MIN", "Val ING max %" := "ANALOGAS"."096PIT005"."ING MAX", "Val ING min %" := "ANALOGAS"."096PIT005"."ING MIN", "OUT ing" => "ANALOGAS"."096PIT005".ESCALIZADA, "OUT %" => "ANALOGAS"."096PIT005".PORCENTAJE)
   END_RUNG
   // the same network as SCL:
   "ESC 4-20mA fail max"(IN := "TRANSMISOR PRESION SUCCION BOMBA 096PIT005",
                         "CD max" := "ANALOGAS"."096PIT005"."CD MAX",
                         "CD min" := "ANALOGAS"."096PIT005"."CD MIN",
                         "Val ING max %" := "ANALOGAS"."096PIT005"."ING MAX",
                         "Val ING min %" := "ANALOGAS"."096PIT005"."ING MIN",
                         "OUT ing" => "ANALOGAS"."096PIT005".ESCALIZADA,
                         "OUT %" => "ANALOGAS"."096PIT005".PORCENTAJE);
END_REGION

REGION Network 2: 096PIT008
   RUNG wire#powerrail
      "ESC 4-20mA fail max"(IN := "TRANSMISOR PRESION DESCARGA BOMBA 096PIT008", "CD max" := "ANALOGAS"."096PIT008"."CD MAX", "CD min" := "ANALOGAS"."096PIT008"."CD MIN", "Val ING max %" := "ANALOGAS"."096PIT008"."ING MAX", "Val ING min %" := "ANALOGAS"."096PIT008"."ING MIN", "OUT ing" => "ANALOGAS"."096PIT008".ESCALIZADA, "OUT %" => "ANALOGAS"."096PIT008".PORCENTAJE)
   END_RUNG
   // the same network as SCL:
   "ESC 4-20mA fail max"(IN := "TRANSMISOR PRESION DESCARGA BOMBA 096PIT008",
                         "CD max" := "ANALOGAS"."096PIT008"."CD MAX",
                         "CD min" := "ANALOGAS"."096PIT008"."CD MIN",
                         "Val ING max %" := "ANALOGAS"."096PIT008"."ING MAX",
                         "Val ING min %" := "ANALOGAS"."096PIT008"."ING MIN",
                         "OUT ing" => "ANALOGAS"."096PIT008".ESCALIZADA,
                         "OUT %" => "ANALOGAS"."096PIT008".PORCENTAJE);
END_REGION

REGION Network 3: 096PIT009
   RUNG wire#powerrail
      "ESC 4-20mA fail max"(IN := "TRANSMISOR PRESION SUCCION BOMBA 096PIT009", "CD max" := "ANALOGAS"."096PIT009"."CD MAX", "CD min" := "ANALOGAS"."096PIT009"."CD MIN", "Val ING max %" := "ANALOGAS"."096PIT009"."ING MAX", "Val ING min %" := "ANALOGAS"."096PIT009"."ING MIN", "OUT ing" => "ANALOGAS"."096PIT009".ESCALIZADA, "OUT %" => "ANALOGAS"."096PIT009".PORCENTAJE)
   END_RUNG
   // the same network as SCL:
   "ESC 4-20mA fail max"(IN := "TRANSMISOR PRESION SUCCION BOMBA 096PIT009",
                         "CD max" := "ANALOGAS"."096PIT009"."CD MAX",
                         "CD min" := "ANALOGAS"."096PIT009"."CD MIN",
                         "Val ING max %" := "ANALOGAS"."096PIT009"."ING MAX",
                         "Val ING min %" := "ANALOGAS"."096PIT009"."ING MIN",
                         "OUT ing" => "ANALOGAS"."096PIT009".ESCALIZADA,
                         "OUT %" => "ANALOGAS"."096PIT009".PORCENTAJE);
END_REGION

REGION Network 4: 096PIT010
   RUNG wire#powerrail
      "ESC 4-20mA fail max"(IN := "TRANSMISOR PRESION DESCARGA BOMBA 096PIT010", "CD max" := "ANALOGAS"."096PIT010"."CD MAX", "CD min" := "ANALOGAS"."096PIT010"."CD MIN", "Val ING max %" := "ANALOGAS"."096PIT010"."ING MAX", "Val ING min %" := "ANALOGAS"."096PIT010"."ING MIN", "OUT ing" => "ANALOGAS"."096PIT010".ESCALIZADA, "OUT %" => "ANALOGAS"."096PIT010".PORCENTAJE)
   END_RUNG
   // the same network as SCL:
   "ESC 4-20mA fail max"(IN := "TRANSMISOR PRESION DESCARGA BOMBA 096PIT010",
                         "CD max" := "ANALOGAS"."096PIT010"."CD MAX",
                         "CD min" := "ANALOGAS"."096PIT010"."CD MIN",
                         "Val ING max %" := "ANALOGAS"."096PIT010"."ING MAX",
                         "Val ING min %" := "ANALOGAS"."096PIT010"."ING MIN",
                         "OUT ing" => "ANALOGAS"."096PIT010".ESCALIZADA,
                         "OUT %" => "ANALOGAS"."096PIT010".PORCENTAJE);
END_REGION

REGION Network 5: 096PIT004
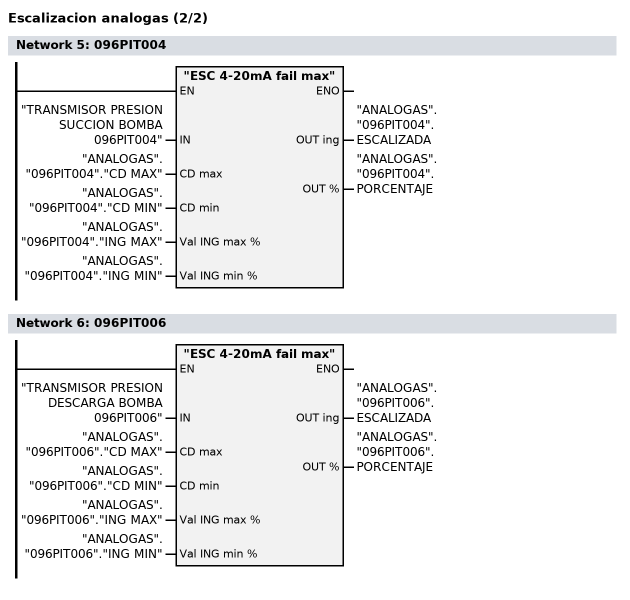
   RUNG wire#powerrail
      "ESC 4-20mA fail max"(IN := "TRANSMISOR PRESION SUCCION BOMBA 096PIT004", "CD max" := "ANALOGAS"."096PIT004"."CD MAX", "CD min" := "ANALOGAS"."096PIT004"."CD MIN", "Val ING max %" := "ANALOGAS"."096PIT004"."ING MAX", "Val ING min %" := "ANALOGAS"."096PIT004"."ING MIN", "OUT ing" => "ANALOGAS"."096PIT004".ESCALIZADA, "OUT %" => "ANALOGAS"."096PIT004".PORCENTAJE)
   END_RUNG
   // the same network as SCL:
   "ESC 4-20mA fail max"(IN := "TRANSMISOR PRESION SUCCION BOMBA 096PIT004",
                         "CD max" := "ANALOGAS"."096PIT004"."CD MAX",
                         "CD min" := "ANALOGAS"."096PIT004"."CD MIN",
                         "Val ING max %" := "ANALOGAS"."096PIT004"."ING MAX",
                         "Val ING min %" := "ANALOGAS"."096PIT004"."ING MIN",
                         "OUT ing" => "ANALOGAS"."096PIT004".ESCALIZADA,
                         "OUT %" => "ANALOGAS"."096PIT004".PORCENTAJE);
END_REGION

REGION Network 6: 096PIT006
   RUNG wire#powerrail
      "ESC 4-20mA fail max"(IN := "TRANSMISOR PRESION DESCARGA BOMBA 096PIT006", "CD max" := "ANALOGAS"."096PIT006"."CD MAX", "CD min" := "ANALOGAS"."096PIT006"."CD MIN", "Val ING max %" := "ANALOGAS"."096PIT006"."ING MAX", "Val ING min %" := "ANALOGAS"."096PIT006"."ING MIN", "OUT ing" => "ANALOGAS"."096PIT006".ESCALIZADA, "OUT %" => "ANALOGAS"."096PIT006".PORCENTAJE)
   END_RUNG
   // the same network as SCL:
   "ESC 4-20mA fail max"(IN := "TRANSMISOR PRESION DESCARGA BOMBA 096PIT006",
                         "CD max" := "ANALOGAS"."096PIT006"."CD MAX",
                         "CD min" := "ANALOGAS"."096PIT006"."CD MIN",
                         "Val ING max %" := "ANALOGAS"."096PIT006"."ING MAX",
                         "Val ING min %" := "ANALOGAS"."096PIT006"."ING MIN",
                         "OUT ing" => "ANALOGAS"."096PIT006".ESCALIZADA,
                         "OUT %" => "ANALOGAS"."096PIT006".PORCENTAJE);
END_REGION
END_FUNCTION

FUNCTION "ARRANQUE MOTORES BIOGAS" : Void   // FC2, LAD
{ S7_Optimized_Access := 'TRUE' }
VERSION : 0.1
   VAR_TEMP
      "Tiempo cumplido B5A" : Bool;
      "Tiempo cumplido B5B" : Bool;
   END_VAR
   VAR_TEMP   // added for the SCL form of the ladder/FBD networks
      _w1 : Bool;
      _w2 : Bool;
      _w3 : Bool;
      _w4 : Bool;
   END_VAR
BEGIN

REGION Network 1: TIEMPO PRESION SUCCION
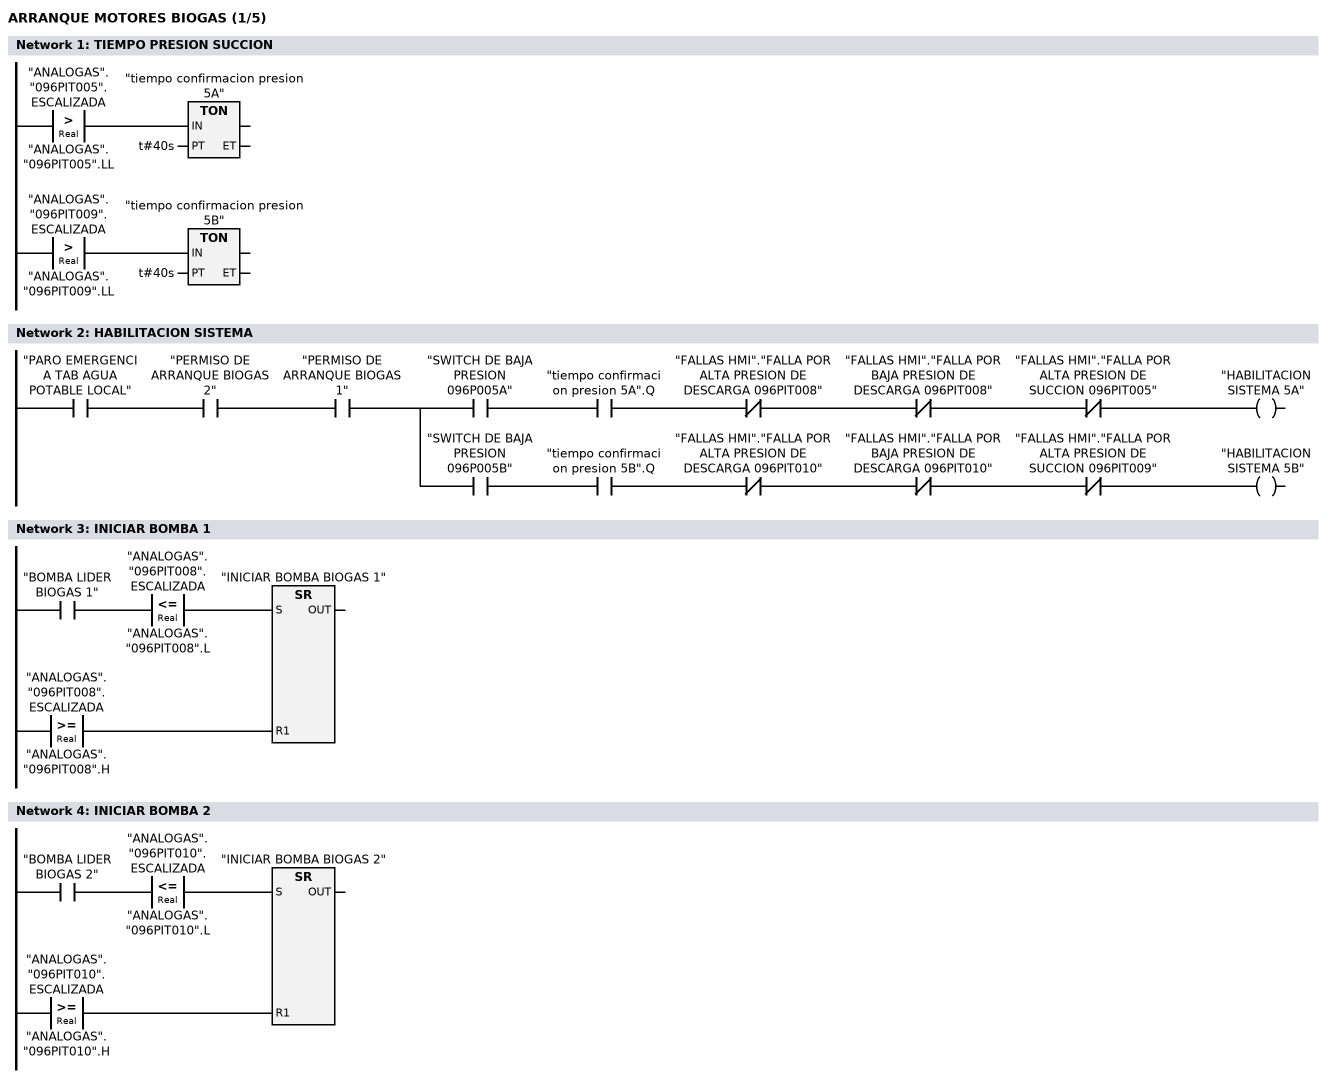
   "tiempo confirmacion presion 5A".TON(IN := "ANALOGAS"."096PIT005".ESCALIZADA > "ANALOGAS"."096PIT005".LL,
                           PT := t#40s);
   "tiempo confirmacion presion 5B".TON(IN := "ANALOGAS"."096PIT009".ESCALIZADA > "ANALOGAS"."096PIT009".LL,
                           PT := t#40s);
END_REGION

REGION Network 2: HABILITACION SISTEMA
   RUNG wire#powerrail
      Contact( "PARO EMERGENCIA TAB AGUA POTABLE LOCAL" )
      Contact( "PERMISO DE ARRANQUE BIOGAS 2" )
      Contact( "PERMISO DE ARRANQUE BIOGAS 1" )
      wire#w1
      Contact( "SWITCH DE BAJA PRESION 096P005A" )
      Contact( "tiempo confirmacion presion 5A".Q )
      I_Contact( "FALLAS HMI"."FALLA POR ALTA PRESION DE DESCARGA 096PIT008" )
      I_Contact( "FALLAS HMI"."FALLA POR BAJA PRESION DE DESCARGA 096PIT008" )
      I_Contact( "FALLAS HMI"."FALLA POR ALTA PRESION DE SUCCION 096PIT005" )
      Coil( "HABILITACION SISTEMA 5A" )
   END_RUNG
   RUNG wire#w1
      Contact( "SWITCH DE BAJA PRESION 096P005B" )
      Contact( "tiempo confirmacion presion 5B".Q )
      I_Contact( "FALLAS HMI"."FALLA POR ALTA PRESION DE DESCARGA 096PIT010" )
      I_Contact( "FALLAS HMI"."FALLA POR BAJA PRESION DE DESCARGA 096PIT010" )
      I_Contact( "FALLAS HMI"."FALLA POR ALTA PRESION DE SUCCION 096PIT009" )
      Coil( "HABILITACION SISTEMA 5B" )
   END_RUNG
   // the same network as SCL:
   #_w1 := "PARO EMERGENCIA TAB AGUA POTABLE LOCAL" AND "PERMISO DE ARRANQUE BIOGAS 2" AND "PERMISO DE ARRANQUE BIOGAS 1";
   "HABILITACION SISTEMA 5A" := #_w1 AND "SWITCH DE BAJA PRESION 096P005A" AND "tiempo confirmacion presion 5A".Q AND NOT "FALLAS HMI"."FALLA POR ALTA PRESION DE DESCARGA 096PIT008" AND NOT "FALLAS HMI"."FALLA POR BAJA PRESION DE DESCARGA 096PIT008" AND NOT "FALLAS HMI"."FALLA POR ALTA PRESION DE SUCCION 096PIT005";
   "HABILITACION SISTEMA 5B" := #_w1 AND "SWITCH DE BAJA PRESION 096P005B" AND "tiempo confirmacion presion 5B".Q AND NOT "FALLAS HMI"."FALLA POR ALTA PRESION DE DESCARGA 096PIT010" AND NOT "FALLAS HMI"."FALLA POR BAJA PRESION DE DESCARGA 096PIT010" AND NOT "FALLAS HMI"."FALLA POR ALTA PRESION DE SUCCION 096PIT009";
END_REGION

REGION Network 3: INICIAR BOMBA 1
   RUNG wire#powerrail
      Contact( "BOMBA LIDER BIOGAS 1" )
      { S7_Templates := "SrcType := Real" } LE_Contact(in1 := "ANALOGAS"."096PIT008".ESCALIZADA, in2 := "ANALOGAS"."096PIT008".L)
      S_SR(operand := "INICIAR BOMBA BIOGAS 1", r1 := wire#w1)
   END_RUNG
   RUNG wire#powerrail
      { S7_Templates := "SrcType := Real" } GE_Contact(in1 := "ANALOGAS"."096PIT008".ESCALIZADA, in2 := "ANALOGAS"."096PIT008".H)
   END_RUNG wire#w1
   // the same network as SCL:
   IF "BOMBA LIDER BIOGAS 1" AND ("ANALOGAS"."096PIT008".ESCALIZADA <= "ANALOGAS"."096PIT008".L) THEN
       "INICIAR BOMBA BIOGAS 1" := TRUE;   // SR flip-flop
   END_IF;
   IF "ANALOGAS"."096PIT008".ESCALIZADA >= "ANALOGAS"."096PIT008".H THEN
       "INICIAR BOMBA BIOGAS 1" := FALSE;
   END_IF;
END_REGION

REGION Network 4: INICIAR BOMBA 2
   RUNG wire#powerrail
      Contact( "BOMBA LIDER BIOGAS 2" )
      { S7_Templates := "SrcType := Real" } LE_Contact(in1 := "ANALOGAS"."096PIT010".ESCALIZADA, in2 := "ANALOGAS"."096PIT010".L)
      S_SR(operand := "INICIAR BOMBA BIOGAS 2", r1 := wire#w1)
   END_RUNG
   RUNG wire#powerrail
      { S7_Templates := "SrcType := Real" } GE_Contact(in1 := "ANALOGAS"."096PIT010".ESCALIZADA, in2 := "ANALOGAS"."096PIT010".H)
   END_RUNG wire#w1
   // the same network as SCL:
   IF "BOMBA LIDER BIOGAS 2" AND ("ANALOGAS"."096PIT010".ESCALIZADA <= "ANALOGAS"."096PIT010".L) THEN
       "INICIAR BOMBA BIOGAS 2" := TRUE;   // SR flip-flop
   END_IF;
   IF "ANALOGAS"."096PIT010".ESCALIZADA >= "ANALOGAS"."096PIT010".H THEN
       "INICIAR BOMBA BIOGAS 2" := FALSE;
   END_IF;
END_REGION

REGION Network 5: ARRANQUE 096P005A
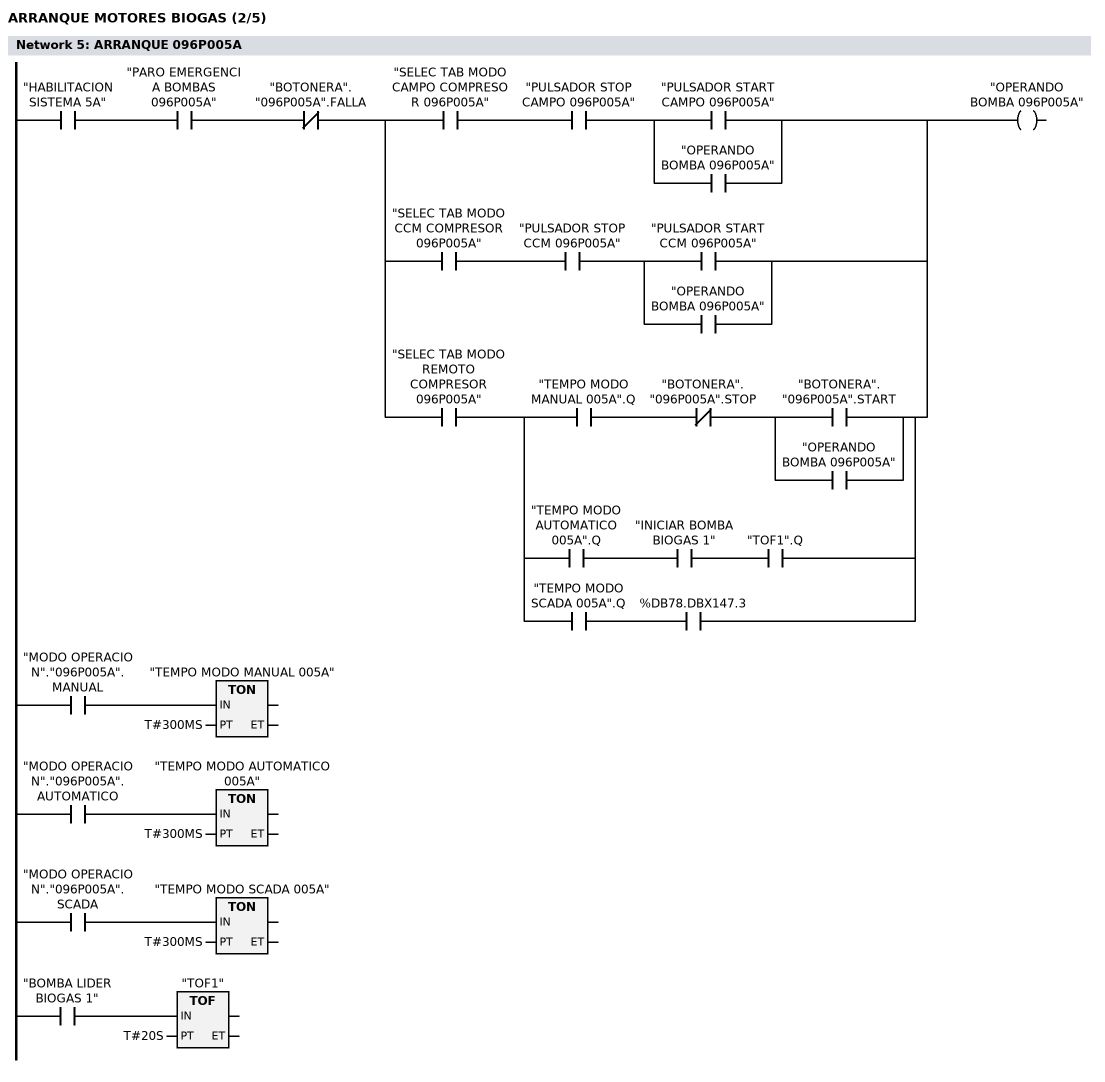
   "OPERANDO BOMBA 096P005A" := "HABILITACION SISTEMA 5A" AND "PARO EMERGENCIA BOMBAS 096P005A" AND NOT "BOTONERA"."096P005A".FALLA AND (("SELEC TAB MODO CAMPO COMPRESOR 096P005A" AND "PULSADOR STOP CAMPO 096P005A" AND ("PULSADOR START CAMPO 096P005A" OR "OPERANDO BOMBA 096P005A")) OR ("SELEC TAB MODO CCM COMPRESOR 096P005A" AND "PULSADOR STOP CCM 096P005A" AND ("PULSADOR START CCM 096P005A" OR "OPERANDO BOMBA 096P005A")) OR ("SELEC TAB MODO REMOTO COMPRESOR 096P005A" AND (("TEMPO MODO MANUAL 005A".Q AND NOT "BOTONERA"."096P005A".STOP AND ("BOTONERA"."096P005A".START OR "OPERANDO BOMBA 096P005A")) OR ("TEMPO MODO AUTOMATICO 005A".Q AND "INICIAR BOMBA BIOGAS 1" AND "TOF1".Q) OR ("TEMPO MODO SCADA 005A".Q AND %DB78.DBX147.3))));
   "TEMPO MODO MANUAL 005A".TON(IN := "MODO OPERACION"."096P005A".MANUAL, PT := T#300MS);
   "TEMPO MODO AUTOMATICO 005A".TON(IN := "MODO OPERACION"."096P005A".AUTOMATICO, PT := T#300MS);
   "TEMPO MODO SCADA 005A".TON(IN := "MODO OPERACION"."096P005A".SCADA, PT := T#300MS);
   "TOF1".TOF(IN := "BOMBA LIDER BIOGAS 1", PT := T#20S);
END_REGION

REGION Network 6: ARRANQUE 096P005B
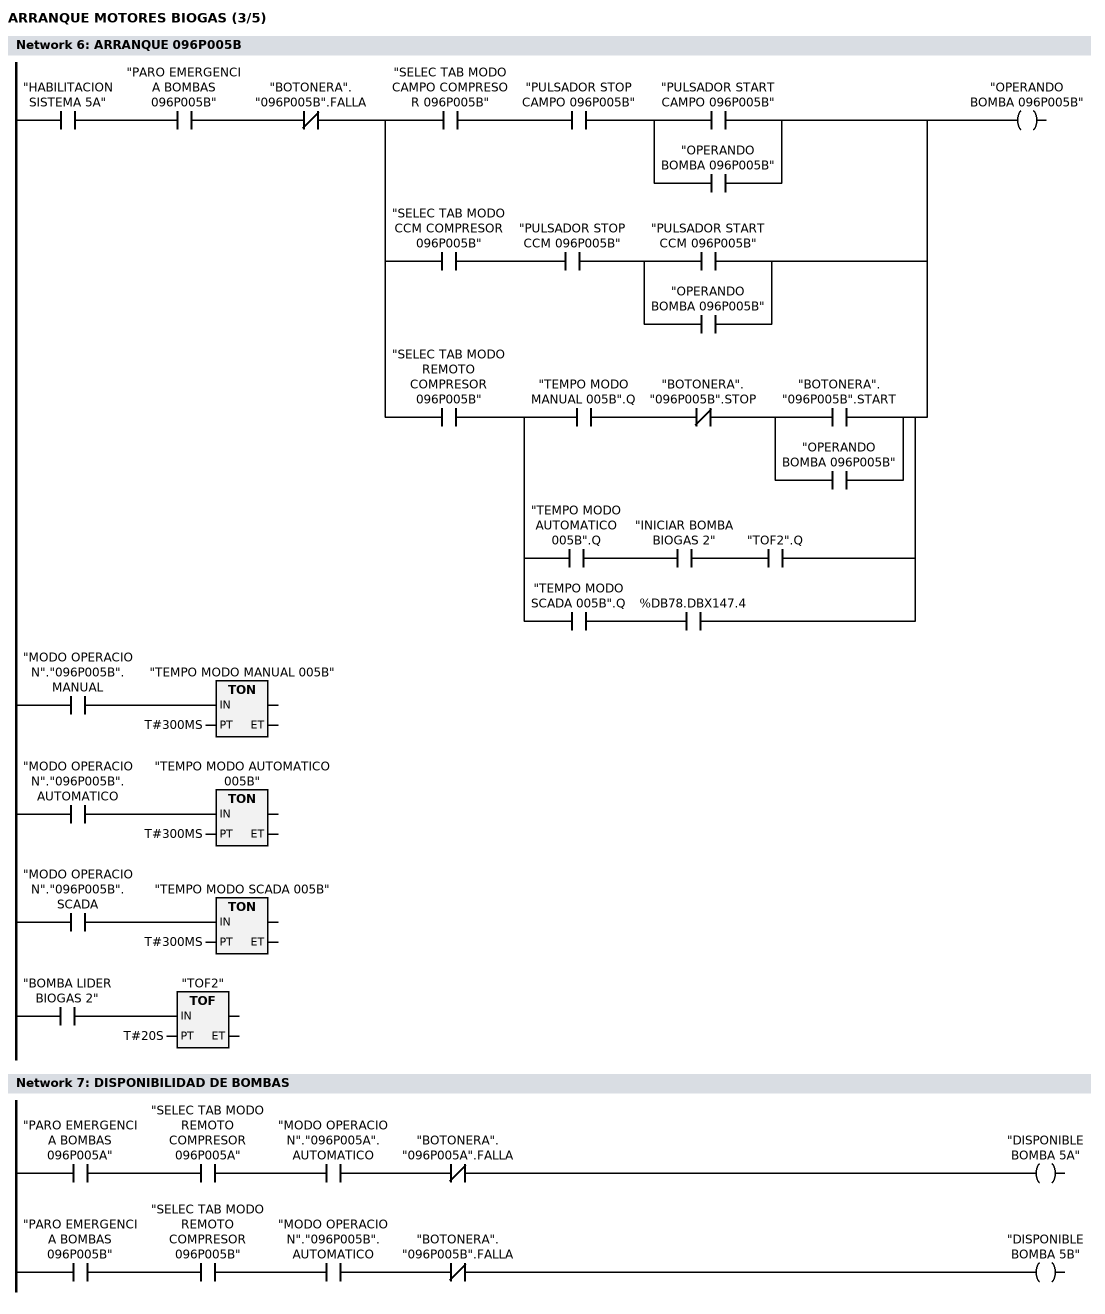
   "OPERANDO BOMBA 096P005B" := "HABILITACION SISTEMA 5A" AND "PARO EMERGENCIA BOMBAS 096P005B" AND NOT "BOTONERA"."096P005B".FALLA AND (("SELEC TAB MODO CAMPO COMPRESOR 096P005B" AND "PULSADOR STOP CAMPO 096P005B" AND ("PULSADOR START CAMPO 096P005B" OR "OPERANDO BOMBA 096P005B")) OR ("SELEC TAB MODO CCM COMPRESOR 096P005B" AND "PULSADOR STOP CCM 096P005B" AND ("PULSADOR START CCM 096P005B" OR "OPERANDO BOMBA 096P005B")) OR ("SELEC TAB MODO REMOTO COMPRESOR 096P005B" AND (("TEMPO MODO MANUAL 005B".Q AND NOT "BOTONERA"."096P005B".STOP AND ("BOTONERA"."096P005B".START OR "OPERANDO BOMBA 096P005B")) OR ("TEMPO MODO AUTOMATICO 005B".Q AND "INICIAR BOMBA BIOGAS 2" AND "TOF2".Q) OR ("TEMPO MODO SCADA 005B".Q AND %DB78.DBX147.4))));
   "TEMPO MODO MANUAL 005B".TON(IN := "MODO OPERACION"."096P005B".MANUAL, PT := T#300MS);
   "TEMPO MODO AUTOMATICO 005B".TON(IN := "MODO OPERACION"."096P005B".AUTOMATICO, PT := T#300MS);
   "TEMPO MODO SCADA 005B".TON(IN := "MODO OPERACION"."096P005B".SCADA, PT := T#300MS);
   "TOF2".TOF(IN := "BOMBA LIDER BIOGAS 2", PT := T#20S);
END_REGION

REGION Network 7: DISPONIBILIDAD DE BOMBAS
   RUNG wire#powerrail
      Contact( "PARO EMERGENCIA BOMBAS 096P005A" )
      Contact( "SELEC TAB MODO REMOTO COMPRESOR 096P005A" )
      Contact( "MODO OPERACION"."096P005A".AUTOMATICO )
      I_Contact( "BOTONERA"."096P005A".FALLA )
      Coil( "DISPONIBLE BOMBA 5A" )
   END_RUNG
   RUNG wire#powerrail
      Contact( "PARO EMERGENCIA BOMBAS 096P005B" )
      Contact( "SELEC TAB MODO REMOTO COMPRESOR 096P005B" )
      Contact( "MODO OPERACION"."096P005B".AUTOMATICO )
      I_Contact( "BOTONERA"."096P005B".FALLA )
      Coil( "DISPONIBLE BOMBA 5B" )
   END_RUNG
   // the same network as SCL:
   "DISPONIBLE BOMBA 5A" := "PARO EMERGENCIA BOMBAS 096P005A" AND "SELEC TAB MODO REMOTO COMPRESOR 096P005A" AND "MODO OPERACION"."096P005A".AUTOMATICO AND NOT "BOTONERA"."096P005A".FALLA;
   "DISPONIBLE BOMBA 5B" := "PARO EMERGENCIA BOMBAS 096P005B" AND "SELEC TAB MODO REMOTO COMPRESOR 096P005B" AND "MODO OPERACION"."096P005B".AUTOMATICO AND NOT "BOTONERA"."096P005B".FALLA;
END_REGION

REGION Network 8: CONTEO BOMBA A
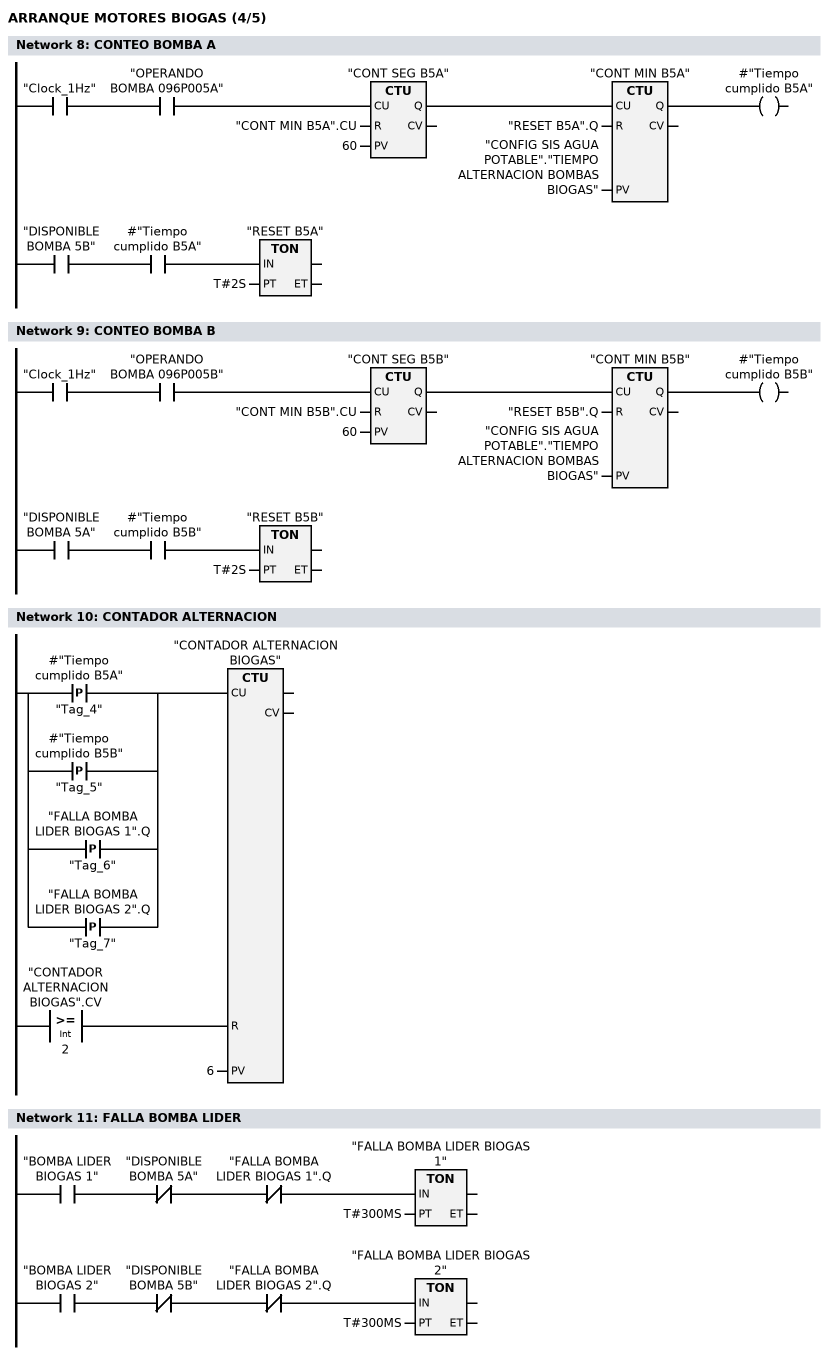
   "CONT SEG B5A".CTU(CU := "Clock_1Hz" AND "OPERANDO BOMBA 096P005A", R := "CONT MIN B5A".CU, PV := 60);
   "CONT MIN B5A".CTU(CU := "CONT SEG B5A".Q,
                      R := "RESET B5A".Q,
                      PV := "CONFIG SIS AGUA POTABLE"."TIEMPO ALTERNACION BOMBAS BIOGAS");
   #"Tiempo cumplido B5A" := "CONT MIN B5A".Q;
   "RESET B5A".TON(IN := "DISPONIBLE BOMBA 5B" AND #"Tiempo cumplido B5A", PT := T#2S);
END_REGION

REGION Network 9: CONTEO BOMBA B
   "CONT SEG B5B".CTU(CU := "Clock_1Hz" AND "OPERANDO BOMBA 096P005B", R := "CONT MIN B5B".CU, PV := 60);
   "CONT MIN B5B".CTU(CU := "CONT SEG B5B".Q,
                      R := "RESET B5B".Q,
                      PV := "CONFIG SIS AGUA POTABLE"."TIEMPO ALTERNACION BOMBAS BIOGAS");
   #"Tiempo cumplido B5B" := "CONT MIN B5B".Q;
   "RESET B5B".TON(IN := "DISPONIBLE BOMBA 5A" AND #"Tiempo cumplido B5B", PT := T#2S);
END_REGION

REGION Network 10: CONTADOR ALTERNACION
   #_w1 := #"Tiempo cumplido B5A" AND NOT "Tag_4";   // rising edge of #"Tiempo cumplido B5A"
   "Tag_4" := #"Tiempo cumplido B5A";
   #_w2 := #"Tiempo cumplido B5B" AND NOT "Tag_5";   // rising edge of #"Tiempo cumplido B5B"
   "Tag_5" := #"Tiempo cumplido B5B";
   #_w3 := "FALLA BOMBA LIDER BIOGAS 1".Q AND NOT "Tag_6";   // rising edge of "FALLA BOMBA LIDER BIOGAS 1".Q
   "Tag_6" := "FALLA BOMBA LIDER BIOGAS 1".Q;
   #_w4 := "FALLA BOMBA LIDER BIOGAS 2".Q AND NOT "Tag_7";   // rising edge of "FALLA BOMBA LIDER BIOGAS 2".Q
   "Tag_7" := "FALLA BOMBA LIDER BIOGAS 2".Q;
   "CONTADOR ALTERNACION BIOGAS".CTU(CU := #_w1 OR #_w2 OR #_w3 OR #_w4,
                           R := "CONTADOR ALTERNACION BIOGAS".CV >= 2,
                           PV := 6);
END_REGION

REGION Network 11: FALLA BOMBA LIDER
   "FALLA BOMBA LIDER BIOGAS 1".TON(IN := "BOMBA LIDER BIOGAS 1" AND NOT "DISPONIBLE BOMBA 5A" AND NOT "FALLA BOMBA LIDER BIOGAS 1".Q,
                           PT := T#300MS);
   "FALLA BOMBA LIDER BIOGAS 2".TON(IN := "BOMBA LIDER BIOGAS 2" AND NOT "DISPONIBLE BOMBA 5B" AND NOT "FALLA BOMBA LIDER BIOGAS 2".Q,
                           PT := T#300MS);
END_REGION

REGION Network 12: BOMBA LIDER
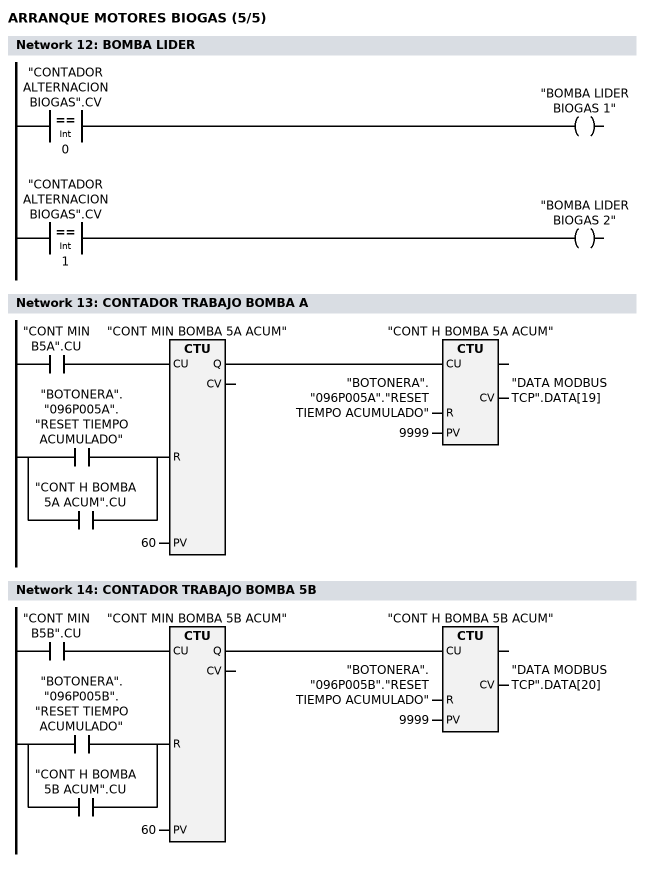
   RUNG wire#powerrail
      { S7_Templates := "SrcType := Int" } EQ_Contact(in1 := "CONTADOR ALTERNACION BIOGAS".CV, in2 := 0)
      Coil( "BOMBA LIDER BIOGAS 1" )
   END_RUNG
   RUNG wire#powerrail
      { S7_Templates := "SrcType := Int" } EQ_Contact(in1 := "CONTADOR ALTERNACION BIOGAS".CV, in2 := 1)
      Coil( "BOMBA LIDER BIOGAS 2" )
   END_RUNG
   // the same network as SCL:
   "BOMBA LIDER BIOGAS 1" := "CONTADOR ALTERNACION BIOGAS".CV = 0;
   "BOMBA LIDER BIOGAS 2" := "CONTADOR ALTERNACION BIOGAS".CV = 1;
END_REGION

REGION Network 13: CONTADOR TRABAJO BOMBA A
   "CONT MIN BOMBA 5A ACUM".CTU(CU := "CONT MIN B5A".CU,
                           R := "BOTONERA"."096P005A"."RESET TIEMPO ACUMULADO" OR "CONT H BOMBA 5A ACUM".CU,
                           PV := 60);
   "CONT H BOMBA 5A ACUM".CTU(CU := "CONT MIN BOMBA 5A ACUM".Q,
                           R := "BOTONERA"."096P005A"."RESET TIEMPO ACUMULADO",
                           PV := 9999,
                           CV => "DATA MODBUS TCP".DATA[19]);
END_REGION

REGION Network 14: CONTADOR TRABAJO BOMBA 5B
   "CONT MIN BOMBA 5B ACUM".CTU(CU := "CONT MIN B5B".CU,
                           R := "BOTONERA"."096P005B"."RESET TIEMPO ACUMULADO" OR "CONT H BOMBA 5B ACUM".CU,
                           PV := 60);
   "CONT H BOMBA 5B ACUM".CTU(CU := "CONT MIN BOMBA 5B ACUM".Q,
                           R := "BOTONERA"."096P005B"."RESET TIEMPO ACUMULADO",
                           PV := 9999,
                           CV => "DATA MODBUS TCP".DATA[20]);
END_REGION
END_FUNCTION

FUNCTION "ESC 4-20mA fail max" : Void   // FC3, LAD
{ S7_Optimized_Access := 'TRUE' }
VERSION : 0.1
   VAR_INPUT
      IN : Word;
      "CD max" : Real;
      "CD min" : Real;
      "Val ING max %" : Real;
      "Val ING min %" : Real;
   END_VAR
   VAR_OUTPUT
      "OUT ing" : Real;
      "OUT %" : Real;
   END_VAR
   VAR_TEMP
      "IN Real" : Real;
      "IN ok" : Real;
      "IN error <" : Bool;
      "IN error >" : Bool;
      "IN ESC" : Real;
      Temp_1 : Int;
   END_VAR
BEGIN

REGION Network 1
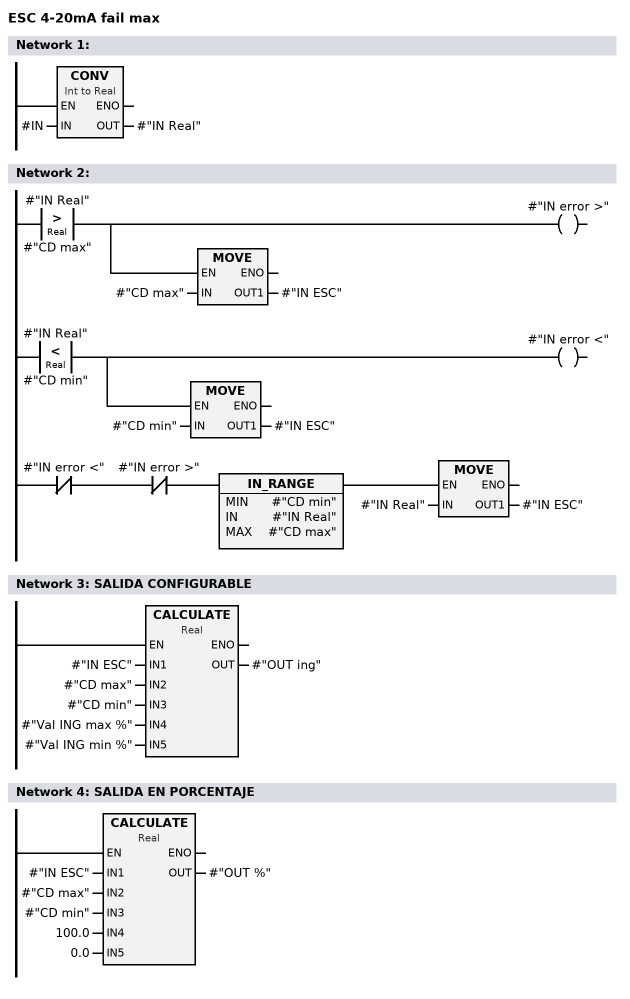
   RUNG wire#powerrail
      { S7_Templates := "[SrcType := Int, DestType := Real]" } Convert(in := #IN, out => #"IN Real")
   END_RUNG
   // the same network as SCL:
   #"IN Real" := INT_TO_REAL(#IN);
END_REGION

REGION Network 2
   RUNG wire#powerrail
      { S7_Templates := "SrcType := Real" } GT_Contact(in1 := #"IN Real", in2 := #"CD max")
      wire#w1
      Coil( #"IN error >" )
   END_RUNG
   RUNG wire#w1
      Move(in := #"CD max", out1 => #"IN ESC")
   END_RUNG
   RUNG wire#powerrail
      { S7_Templates := "SrcType := Real" } LT_Contact(in1 := #"IN Real", in2 := #"CD min")
      wire#w2
      Coil( #"IN error <" )
   END_RUNG
   RUNG wire#w2
      Move(in := #"CD min", out1 => #"IN ESC")
   END_RUNG
   RUNG wire#powerrail
      I_Contact( #"IN error <" )
      I_Contact( #"IN error >" )
      { S7_Templates := "SrcType := Real" } InRange(min := #"CD min", in := #"IN Real", max := #"CD max")
      Move(in := #"IN Real", out1 => #"IN ESC")
   END_RUNG
   // the same network as SCL:
   #"IN error >" := #"IN Real" > #"CD max";
   IF #"IN error >" THEN #"IN ESC" := #"CD max"; END_IF;
   #"IN error <" := #"IN Real" < #"CD min";
   IF #"IN error <" THEN #"IN ESC" := #"CD min"; END_IF;
   IF NOT #"IN error <" AND NOT #"IN error >" AND (#"CD min" <= #"IN Real") AND (#"IN Real" <= #"CD max") THEN
       #"IN ESC" := #"IN Real";
   END_IF;
END_REGION

REGION Network 3: SALIDA CONFIGURABLE
   RUNG wire#powerrail
      { S7_Templates := "SrcType := Real"; S7_Expression := "(((in4-in5)/(in2-in3))*in1)+(in5-(((in4-in5)/(in2-in3))*in3))" } Calculate(in1 := #"IN ESC", in2 := #"CD max", in3 := #"CD min", in4 := #"Val ING max %", in5 := #"Val ING min %", out => #"OUT ing")
   END_RUNG
   // the same network as SCL:
   #"OUT ing" := (((#"Val ING max %"-#"Val ING min %")/(#"CD max"-#"CD min"))*#"IN ESC")+(#"Val ING min %"-(((#"Val ING max %"-#"Val ING min %")/(#"CD max"-#"CD min"))*#"CD min"));
END_REGION

REGION Network 4: SALIDA EN PORCENTAJE
   RUNG wire#powerrail
      { S7_Templates := "SrcType := Real"; S7_Expression := "(((in4-in5)/(in2-in3))*in1)+(in5-(((in4-in5)/(in2-in3))*in3))" } Calculate(in1 := #"IN ESC", in2 := #"CD max", in3 := #"CD min", in4 := 100.0, in5 := 0.0, out => #"OUT %")
   END_RUNG
   // the same network as SCL:
   #"OUT %" := (((100.0-0.0)/(#"CD max"-#"CD min"))*#"IN ESC")+(0.0-(((100.0-0.0)/(#"CD max"-#"CD min"))*#"CD min"));
END_REGION

REGION Network 5: SALIDA EN mA
END_REGION
END_FUNCTION

FUNCTION "COMUNICACION MODBUS CLIENT" : Void   // FC4, LAD
{ S7_Optimized_Access := 'TRUE' }
VERSION : 0.1
BEGIN

REGION Network 1: AS7 - COMM
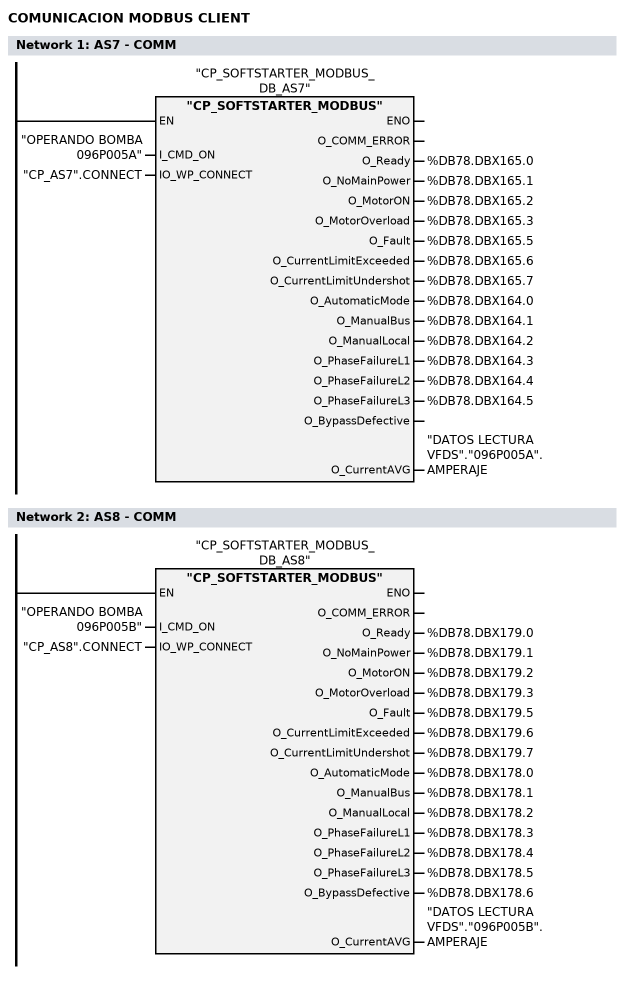
   RUNG wire#powerrail
      "CP_SOFTSTARTER_MODBUS_DB_AS7"(I_CMD_ON := "OPERANDO BOMBA 096P005A", IO_WP_CONNECT := "CP_AS7".CONNECT, O_COMM_ERROR =>, O_Ready => %DB78.DBX165.0, O_NoMainPower => %DB78.DBX165.1, O_MotorON => %DB78.DBX165.2, O_MotorOverload => %DB78.DBX165.3, O_Fault => %DB78.DBX165.5, O_CurrentLimitExceeded => %DB78.DBX165.6, O_CurrentLimitUndershot => %DB78.DBX165.7, O_AutomaticMode => %DB78.DBX164.0, O_ManualBus => %DB78.DBX164.1, O_ManualLocal => %DB78.DBX164.2, O_PhaseFailureL1 => %DB78.DBX164.3, O_PhaseFailureL2 => %DB78.DBX164.4, O_PhaseFailureL3 => %DB78.DBX164.5, O_BypassDefective =>, O_CurrentAVG => "DATOS LECTURA VFDS"."096P005A".AMPERAJE)
   END_RUNG
   // the same network as SCL:
   "CP_SOFTSTARTER_MODBUS_DB_AS7"(I_CMD_ON := "OPERANDO BOMBA 096P005A",   // "CP_SOFTSTARTER_MODBUS"
                           IO_WP_CONNECT := "CP_AS7".CONNECT,
                           O_Ready => %DB78.DBX165.0,
                           O_NoMainPower => %DB78.DBX165.1,
                           O_MotorON => %DB78.DBX165.2,
                           O_MotorOverload => %DB78.DBX165.3,
                           O_Fault => %DB78.DBX165.5,
                           O_CurrentLimitExceeded => %DB78.DBX165.6,
                           O_CurrentLimitUndershot => %DB78.DBX165.7,
                           O_AutomaticMode => %DB78.DBX164.0,
                           O_ManualBus => %DB78.DBX164.1,
                           O_ManualLocal => %DB78.DBX164.2,
                           O_PhaseFailureL1 => %DB78.DBX164.3,
                           O_PhaseFailureL2 => %DB78.DBX164.4,
                           O_PhaseFailureL3 => %DB78.DBX164.5,
                           O_CurrentAVG => "DATOS LECTURA VFDS"."096P005A".AMPERAJE);
END_REGION

REGION Network 2: AS8 - COMM
   RUNG wire#powerrail
      "CP_SOFTSTARTER_MODBUS_DB_AS8"(I_CMD_ON := "OPERANDO BOMBA 096P005B", IO_WP_CONNECT := "CP_AS8".CONNECT, O_COMM_ERROR =>, O_Ready => %DB78.DBX179.0, O_NoMainPower => %DB78.DBX179.1, O_MotorON => %DB78.DBX179.2, O_MotorOverload => %DB78.DBX179.3, O_Fault => %DB78.DBX179.5, O_CurrentLimitExceeded => %DB78.DBX179.6, O_CurrentLimitUndershot => %DB78.DBX179.7, O_AutomaticMode => %DB78.DBX178.0, O_ManualBus => %DB78.DBX178.1, O_ManualLocal => %DB78.DBX178.2, O_PhaseFailureL1 => %DB78.DBX178.3, O_PhaseFailureL2 => %DB78.DBX178.4, O_PhaseFailureL3 => %DB78.DBX178.5, O_BypassDefective => %DB78.DBX178.6, O_CurrentAVG => "DATOS LECTURA VFDS"."096P005B".AMPERAJE)
   END_RUNG
   // the same network as SCL:
   "CP_SOFTSTARTER_MODBUS_DB_AS8"(I_CMD_ON := "OPERANDO BOMBA 096P005B",   // "CP_SOFTSTARTER_MODBUS"
                           IO_WP_CONNECT := "CP_AS8".CONNECT,
                           O_Ready => %DB78.DBX179.0,
                           O_NoMainPower => %DB78.DBX179.1,
                           O_MotorON => %DB78.DBX179.2,
                           O_MotorOverload => %DB78.DBX179.3,
                           O_Fault => %DB78.DBX179.5,
                           O_CurrentLimitExceeded => %DB78.DBX179.6,
                           O_CurrentLimitUndershot => %DB78.DBX179.7,
                           O_AutomaticMode => %DB78.DBX178.0,
                           O_ManualBus => %DB78.DBX178.1,
                           O_ManualLocal => %DB78.DBX178.2,
                           O_PhaseFailureL1 => %DB78.DBX178.3,
                           O_PhaseFailureL2 => %DB78.DBX178.4,
                           O_PhaseFailureL3 => %DB78.DBX178.5,
                           O_BypassDefective => %DB78.DBX178.6,
                           O_CurrentAVG => "DATOS LECTURA VFDS"."096P005B".AMPERAJE);
END_REGION
END_FUNCTION

FUNCTION "ARRANQUE MOTORES AGUA POTABLE" : Void   // FC5, LAD
{ S7_Optimized_Access := 'TRUE' }
VERSION : 0.1
   VAR_TEMP
      "SIN FLUJO SISTEMA 096P001A" : Bool;
      "SIN FLUJO SISTEMA 096P001B" : Bool;
      "SIN FLUJO SISTEMA 096P001C" : Bool;
      "SIN FLUJO SISTEMA 096P001D" : Bool;
      "SIN FLUJO SISTEMA 096P001E" : Bool;
      "SIN FLUJO SISTEMA 096P001F" : Bool;
   END_VAR
BEGIN

REGION Network 1
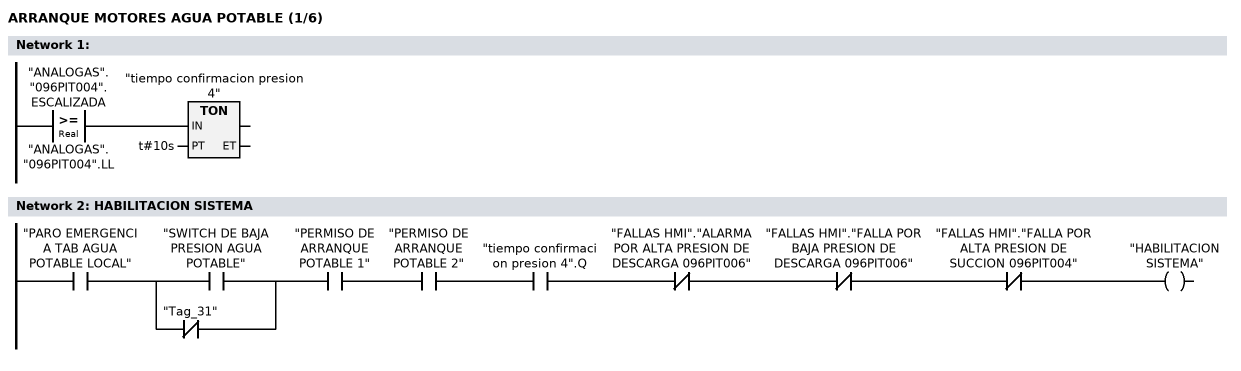
   "tiempo confirmacion presion 4".TON(IN := "ANALOGAS"."096PIT004".ESCALIZADA >= "ANALOGAS"."096PIT004".LL,
                           PT := t#10s);
END_REGION

REGION Network 2: HABILITACION SISTEMA
   RUNG wire#powerrail
      Contact( "PARO EMERGENCIA TAB AGUA POTABLE LOCAL" )
      wire#w1
      Contact( "SWITCH DE BAJA PRESION AGUA POTABLE" )
      wire#w2
      Contact( "PERMISO DE ARRANQUE POTABLE 1" )
      Contact( "PERMISO DE ARRANQUE POTABLE 2" )
      Contact( "tiempo confirmacion presion 4".Q )
      I_Contact( "FALLAS HMI"."ALARMA POR ALTA PRESION DE DESCARGA 096PIT006" )
      I_Contact( "FALLAS HMI"."FALLA POR BAJA PRESION DE DESCARGA 096PIT006" )
      I_Contact( "FALLAS HMI"."FALLA POR ALTA PRESION DE SUCCION 096PIT004" )
      Coil( "HABILITACION SISTEMA" )
   END_RUNG
   RUNG wire#w1
      I_Contact( "Tag_31" )
   END_RUNG wire#w2
   // the same network as SCL:
   "HABILITACION SISTEMA" := "PARO EMERGENCIA TAB AGUA POTABLE LOCAL" AND ("SWITCH DE BAJA PRESION AGUA POTABLE" OR NOT "Tag_31") AND "PERMISO DE ARRANQUE POTABLE 1" AND "PERMISO DE ARRANQUE POTABLE 2" AND "tiempo confirmacion presion 4".Q AND NOT "FALLAS HMI"."ALARMA POR ALTA PRESION DE DESCARGA 096PIT006" AND NOT "FALLAS HMI"."FALLA POR BAJA PRESION DE DESCARGA 096PIT006" AND NOT "FALLAS HMI"."FALLA POR ALTA PRESION DE SUCCION 096PIT004";
END_REGION

REGION Network 3: ARRANQUE 096P004A
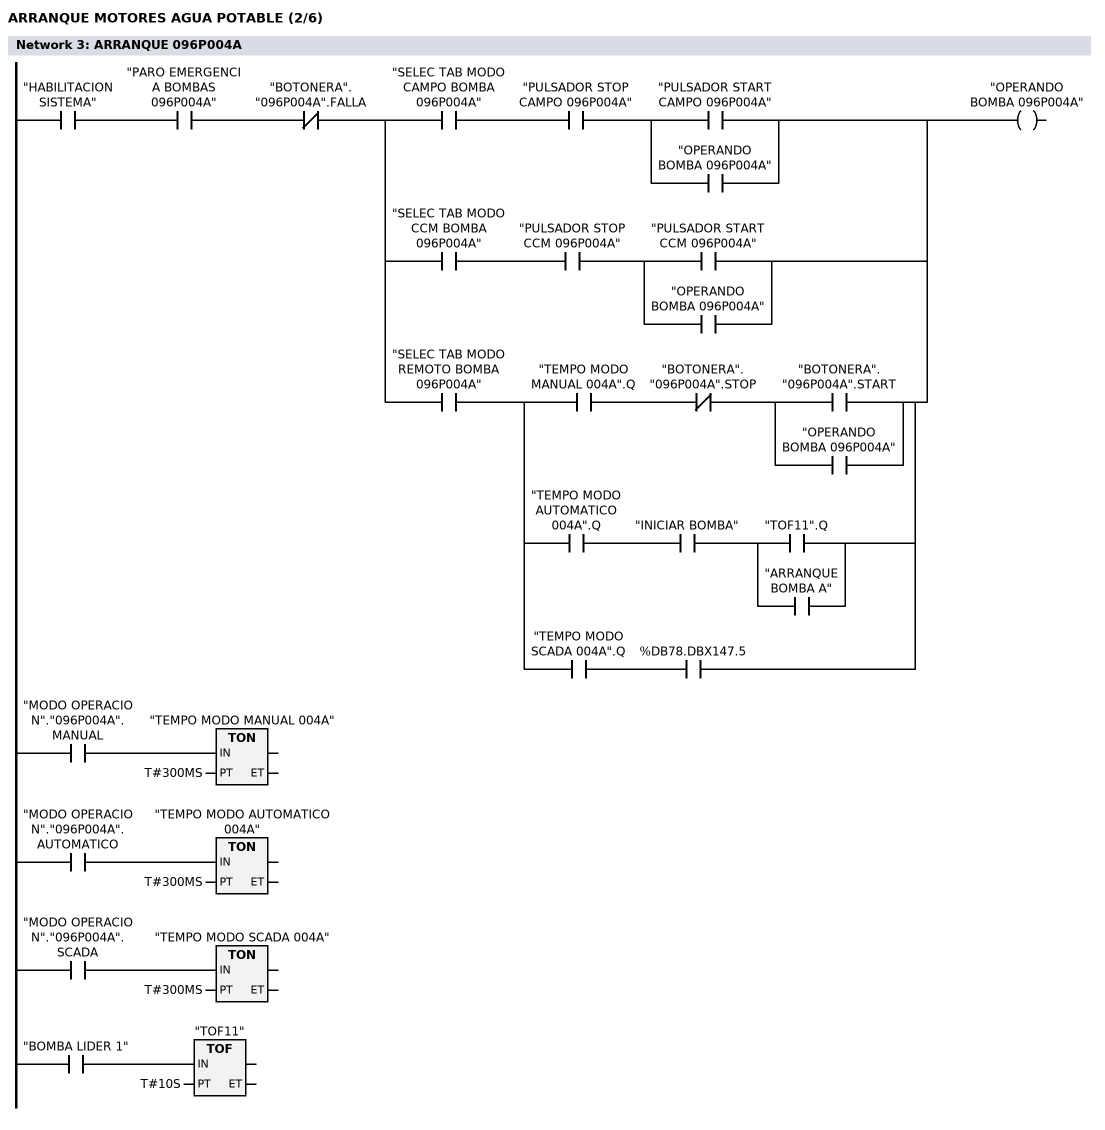
   "OPERANDO BOMBA 096P004A" := "HABILITACION SISTEMA" AND "PARO EMERGENCIA BOMBAS 096P004A" AND NOT "BOTONERA"."096P004A".FALLA AND (("SELEC TAB MODO CAMPO BOMBA 096P004A" AND "PULSADOR STOP CAMPO 096P004A" AND ("PULSADOR START CAMPO 096P004A" OR "OPERANDO BOMBA 096P004A")) OR ("SELEC TAB MODO CCM BOMBA 096P004A" AND "PULSADOR STOP CCM 096P004A" AND ("PULSADOR START CCM 096P004A" OR "OPERANDO BOMBA 096P004A")) OR ("SELEC TAB MODO REMOTO BOMBA 096P004A" AND (("TEMPO MODO MANUAL 004A".Q AND NOT "BOTONERA"."096P004A".STOP AND ("BOTONERA"."096P004A".START OR "OPERANDO BOMBA 096P004A")) OR ("TEMPO MODO AUTOMATICO 004A".Q AND "INICIAR BOMBA" AND ("TOF11".Q OR "ARRANQUE BOMBA A")) OR ("TEMPO MODO SCADA 004A".Q AND %DB78.DBX147.5))));
   "TEMPO MODO MANUAL 004A".TON(IN := "MODO OPERACION"."096P004A".MANUAL, PT := T#300MS);
   "TEMPO MODO AUTOMATICO 004A".TON(IN := "MODO OPERACION"."096P004A".AUTOMATICO, PT := T#300MS);
   "TEMPO MODO SCADA 004A".TON(IN := "MODO OPERACION"."096P004A".SCADA, PT := T#300MS);
   "TOF11".TOF(IN := "BOMBA LIDER 1", PT := T#10S);
END_REGION

REGION Network 4: ARRANQUE 096P004B
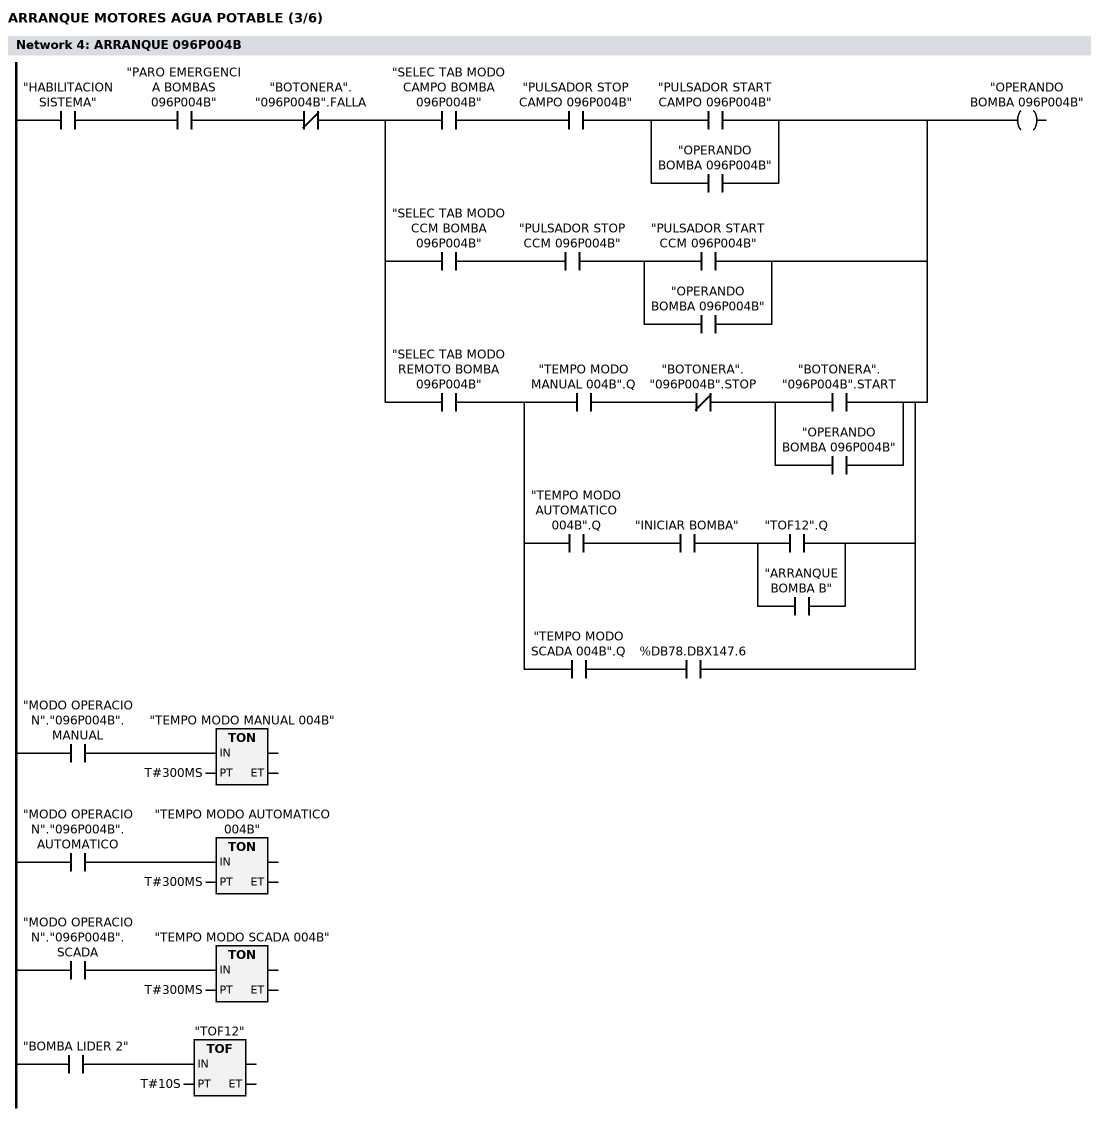
   "OPERANDO BOMBA 096P004B" := "HABILITACION SISTEMA" AND "PARO EMERGENCIA BOMBAS 096P004B" AND NOT "BOTONERA"."096P004B".FALLA AND (("SELEC TAB MODO CAMPO BOMBA 096P004B" AND "PULSADOR STOP CAMPO 096P004B" AND ("PULSADOR START CAMPO 096P004B" OR "OPERANDO BOMBA 096P004B")) OR ("SELEC TAB MODO CCM BOMBA 096P004B" AND "PULSADOR STOP CCM 096P004B" AND ("PULSADOR START CCM 096P004B" OR "OPERANDO BOMBA 096P004B")) OR ("SELEC TAB MODO REMOTO BOMBA 096P004B" AND (("TEMPO MODO MANUAL 004B".Q AND NOT "BOTONERA"."096P004B".STOP AND ("BOTONERA"."096P004B".START OR "OPERANDO BOMBA 096P004B")) OR ("TEMPO MODO AUTOMATICO 004B".Q AND "INICIAR BOMBA" AND ("TOF12".Q OR "ARRANQUE BOMBA B")) OR ("TEMPO MODO SCADA 004B".Q AND %DB78.DBX147.6))));
   "TEMPO MODO MANUAL 004B".TON(IN := "MODO OPERACION"."096P004B".MANUAL, PT := T#300MS);
   "TEMPO MODO AUTOMATICO 004B".TON(IN := "MODO OPERACION"."096P004B".AUTOMATICO, PT := T#300MS);
   "TEMPO MODO SCADA 004B".TON(IN := "MODO OPERACION"."096P004B".SCADA, PT := T#300MS);
   "TOF12".TOF(IN := "BOMBA LIDER 2", PT := T#10S);
END_REGION

REGION Network 5: ARRANQUE 096P004C
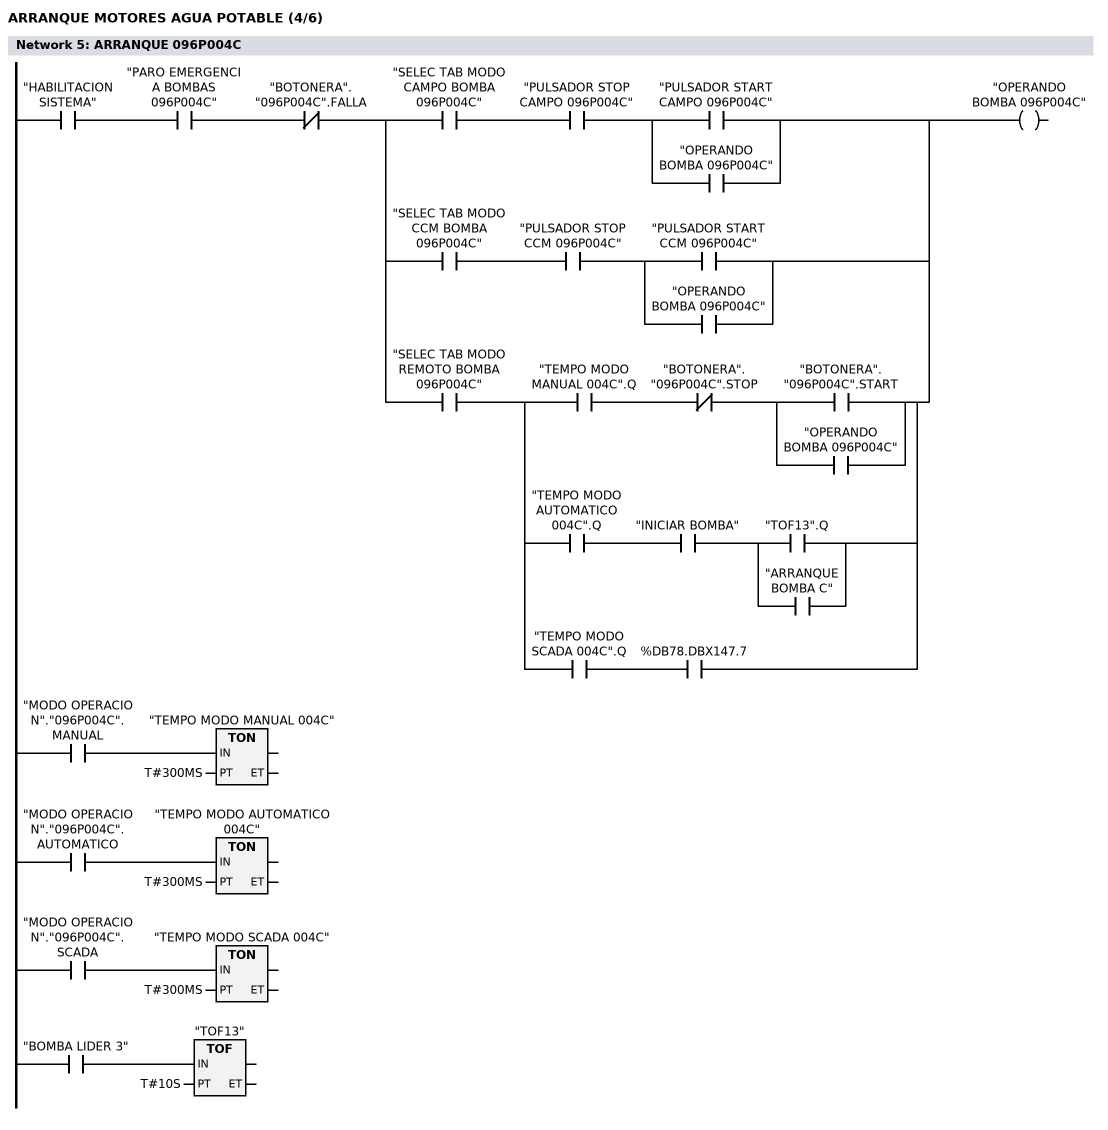
   "OPERANDO BOMBA 096P004C" := "HABILITACION SISTEMA" AND "PARO EMERGENCIA BOMBAS 096P004C" AND NOT "BOTONERA"."096P004C".FALLA AND (("SELEC TAB MODO CAMPO BOMBA 096P004C" AND "PULSADOR STOP CAMPO 096P004C" AND ("PULSADOR START CAMPO 096P004C" OR "OPERANDO BOMBA 096P004C")) OR ("SELEC TAB MODO CCM BOMBA 096P004C" AND "PULSADOR STOP CCM 096P004C" AND ("PULSADOR START CCM 096P004C" OR "OPERANDO BOMBA 096P004C")) OR ("SELEC TAB MODO REMOTO BOMBA 096P004C" AND (("TEMPO MODO MANUAL 004C".Q AND NOT "BOTONERA"."096P004C".STOP AND ("BOTONERA"."096P004C".START OR "OPERANDO BOMBA 096P004C")) OR ("TEMPO MODO AUTOMATICO 004C".Q AND "INICIAR BOMBA" AND ("TOF13".Q OR "ARRANQUE BOMBA C")) OR ("TEMPO MODO SCADA 004C".Q AND %DB78.DBX147.7))));
   "TEMPO MODO MANUAL 004C".TON(IN := "MODO OPERACION"."096P004C".MANUAL, PT := T#300MS);
   "TEMPO MODO AUTOMATICO 004C".TON(IN := "MODO OPERACION"."096P004C".AUTOMATICO, PT := T#300MS);
   "TEMPO MODO SCADA 004C".TON(IN := "MODO OPERACION"."096P004C".SCADA, PT := T#300MS);
   "TOF13".TOF(IN := "BOMBA LIDER 3", PT := T#10S);
END_REGION

REGION Network 6: ARRANQUE 096P004D
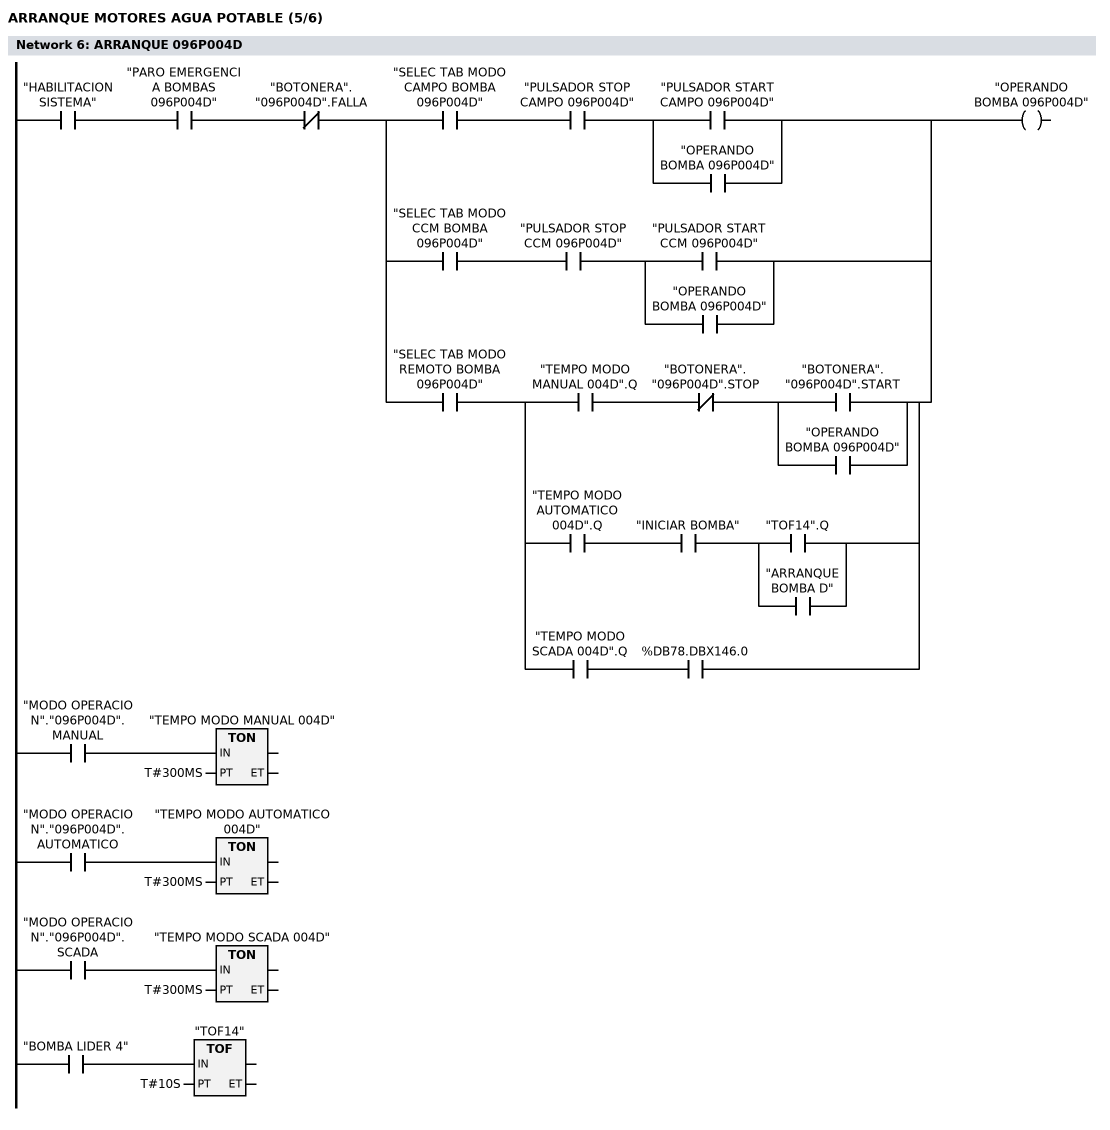
   "OPERANDO BOMBA 096P004D" := "HABILITACION SISTEMA" AND "PARO EMERGENCIA BOMBAS 096P004D" AND NOT "BOTONERA"."096P004D".FALLA AND (("SELEC TAB MODO CAMPO BOMBA 096P004D" AND "PULSADOR STOP CAMPO 096P004D" AND ("PULSADOR START CAMPO 096P004D" OR "OPERANDO BOMBA 096P004D")) OR ("SELEC TAB MODO CCM BOMBA 096P004D" AND "PULSADOR STOP CCM 096P004D" AND ("PULSADOR START CCM 096P004D" OR "OPERANDO BOMBA 096P004D")) OR ("SELEC TAB MODO REMOTO BOMBA 096P004D" AND (("TEMPO MODO MANUAL 004D".Q AND NOT "BOTONERA"."096P004D".STOP AND ("BOTONERA"."096P004D".START OR "OPERANDO BOMBA 096P004D")) OR ("TEMPO MODO AUTOMATICO 004D".Q AND "INICIAR BOMBA" AND ("TOF14".Q OR "ARRANQUE BOMBA D")) OR ("TEMPO MODO SCADA 004D".Q AND %DB78.DBX146.0))));
   "TEMPO MODO MANUAL 004D".TON(IN := "MODO OPERACION"."096P004D".MANUAL, PT := T#300MS);
   "TEMPO MODO AUTOMATICO 004D".TON(IN := "MODO OPERACION"."096P004D".AUTOMATICO, PT := T#300MS);
   "TEMPO MODO SCADA 004D".TON(IN := "MODO OPERACION"."096P004D".SCADA, PT := T#300MS);
   "TOF14".TOF(IN := "BOMBA LIDER 4", PT := T#10S);
END_REGION

REGION Network 7: DISPONIBILIDAD DE BOMBAS
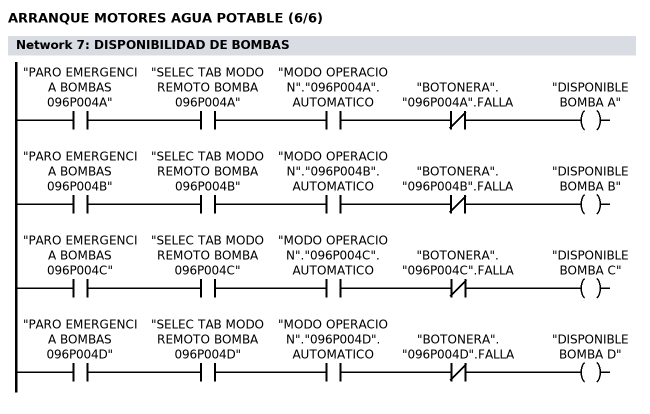
   RUNG wire#powerrail
      Contact( "PARO EMERGENCIA BOMBAS 096P004A" )
      Contact( "SELEC TAB MODO REMOTO BOMBA 096P004A" )
      Contact( "MODO OPERACION"."096P004A".AUTOMATICO )
      I_Contact( "BOTONERA"."096P004A".FALLA )
      Coil( "DISPONIBLE BOMBA A" )
   END_RUNG
   RUNG wire#powerrail
      Contact( "PARO EMERGENCIA BOMBAS 096P004B" )
      Contact( "SELEC TAB MODO REMOTO BOMBA 096P004B" )
      Contact( "MODO OPERACION"."096P004B".AUTOMATICO )
      I_Contact( "BOTONERA"."096P004B".FALLA )
      Coil( "DISPONIBLE BOMBA B" )
   END_RUNG
   RUNG wire#powerrail
      Contact( "PARO EMERGENCIA BOMBAS 096P004C" )
      Contact( "SELEC TAB MODO REMOTO BOMBA 096P004C" )
      Contact( "MODO OPERACION"."096P004C".AUTOMATICO )
      I_Contact( "BOTONERA"."096P004C".FALLA )
      Coil( "DISPONIBLE BOMBA C" )
   END_RUNG
   RUNG wire#powerrail
      Contact( "PARO EMERGENCIA BOMBAS 096P004D" )
      Contact( "SELEC TAB MODO REMOTO BOMBA 096P004D" )
      Contact( "MODO OPERACION"."096P004D".AUTOMATICO )
      I_Contact( "BOTONERA"."096P004D".FALLA )
      Coil( "DISPONIBLE BOMBA D" )
   END_RUNG
   // the same network as SCL:
   "DISPONIBLE BOMBA A" := "PARO EMERGENCIA BOMBAS 096P004A" AND "SELEC TAB MODO REMOTO BOMBA 096P004A" AND "MODO OPERACION"."096P004A".AUTOMATICO AND NOT "BOTONERA"."096P004A".FALLA;
   "DISPONIBLE BOMBA B" := "PARO EMERGENCIA BOMBAS 096P004B" AND "SELEC TAB MODO REMOTO BOMBA 096P004B" AND "MODO OPERACION"."096P004B".AUTOMATICO AND NOT "BOTONERA"."096P004B".FALLA;
   "DISPONIBLE BOMBA C" := "PARO EMERGENCIA BOMBAS 096P004C" AND "SELEC TAB MODO REMOTO BOMBA 096P004C" AND "MODO OPERACION"."096P004C".AUTOMATICO AND NOT "BOTONERA"."096P004C".FALLA;
   "DISPONIBLE BOMBA D" := "PARO EMERGENCIA BOMBAS 096P004D" AND "SELEC TAB MODO REMOTO BOMBA 096P004D" AND "MODO OPERACION"."096P004D".AUTOMATICO AND NOT "BOTONERA"."096P004D".FALLA;
END_REGION
END_FUNCTION

FUNCTION "SISTEMA DE PRESION" : Void   // FC6, LAD
{ S7_Optimized_Access := 'TRUE' }
VERSION : 0.1
   VAR_TEMP
      T1 : Real;
      T2 : Real;
      T3 : Real;
      T4 : Real;
      T5 : Real;
      T6 : Real;
      t7 : Real;
      "Tiempo 1" : DInt;
      "Tiempo 2" : DInt;
      "Tiempo 3" : DInt;
      "Tiempo 4" : DInt;
      "Tiempo 5" : DInt;
      "Tiempo 6" : DInt;
      "Tiempo 7" : DInt;
      "DIFERENCIAL ARRANQUE" : Real;
      "DIFERENCIAL DORMIR" : Real;
      "FRECUENCIA OPERACION" : Real;
      ADICION : Bool;
      ACTIVAR : Bool;
      "SIN BOMBAS" : Bool;
      "Tiempo cumplido B1" : Bool;
      "Tiempo cumplido B2" : Bool;
      "Tiempo cumplido B3" : Bool;
      "Tiempo cumplido B4" : Bool;
      "Tiempo cumplido B5" : Bool;
      "Tiempo cumplido B6" : Bool;
      TEST1 : Bool;
      TEST2 : Bool;
      TEST3 : Bool;
      TEST4 : Bool;
      TEST5 : Bool;
      TEST6 : Bool;
      TEST7 : Bool;
      TEST8 : Bool;
      TEST9 : Bool;
      TEST10 : Bool;
      TEST11 : Bool;
      TEST12 : Bool;
   END_VAR
   VAR_TEMP   // added for the SCL form of the ladder/FBD networks
      _w1 : Bool;
      _w2 : Bool;
      _w3 : Bool;
      _w4 : Bool;
      _w5 : Bool;
      _w6 : Bool;
      _w7 : Bool;
      _w8 : Bool;
   END_VAR
BEGIN

REGION Network 1: convertir temporizadores
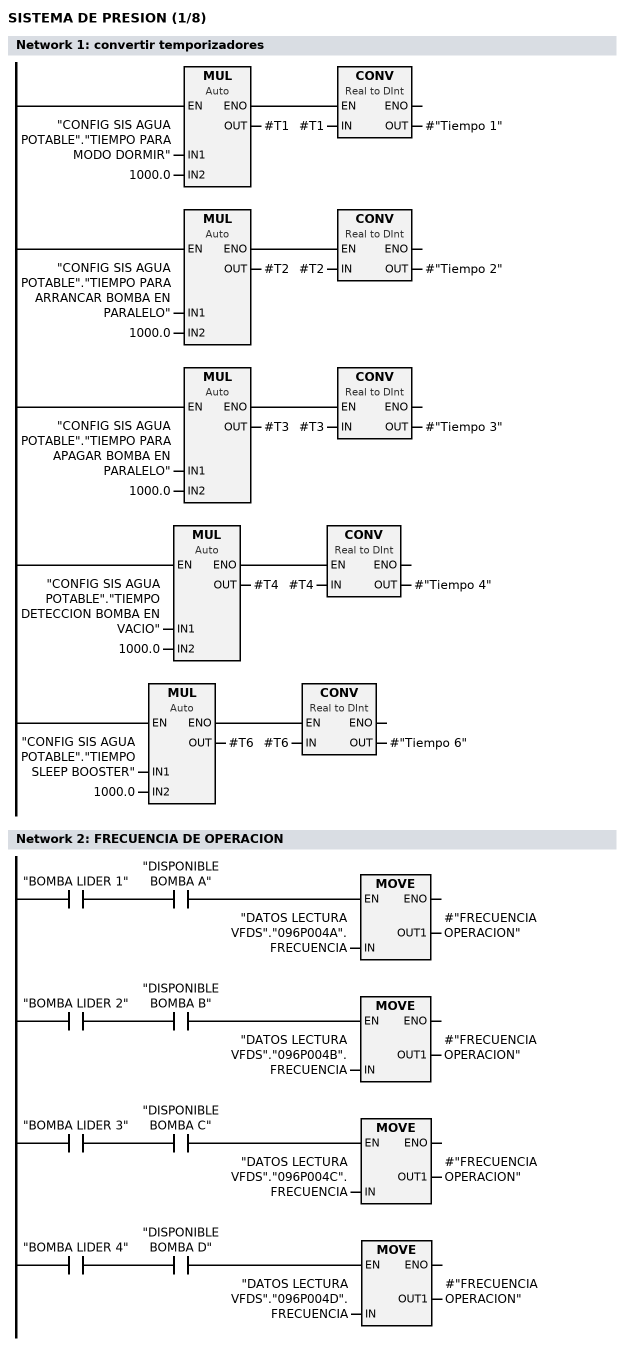
   RUNG wire#powerrail
      Mul(in1 := "CONFIG SIS AGUA POTABLE"."TIEMPO PARA MODO DORMIR", in2 := 1000.0, out => #T1)
      { S7_Templates := "[SrcType := Real, DestType := DInt]" } Convert(in := #T1, out => #"Tiempo 1")
   END_RUNG
   RUNG wire#powerrail
      Mul(in1 := "CONFIG SIS AGUA POTABLE"."TIEMPO PARA ARRANCAR BOMBA EN PARALELO", in2 := 1000.0, out => #T2)
      { S7_Templates := "[SrcType := Real, DestType := DInt]" } Convert(in := #T2, out => #"Tiempo 2")
   END_RUNG
   RUNG wire#powerrail
      Mul(in1 := "CONFIG SIS AGUA POTABLE"."TIEMPO PARA APAGAR BOMBA EN PARALELO", in2 := 1000.0, out => #T3)
      { S7_Templates := "[SrcType := Real, DestType := DInt]" } Convert(in := #T3, out => #"Tiempo 3")
   END_RUNG
   RUNG wire#powerrail
      Mul(in1 := "CONFIG SIS AGUA POTABLE"."TIEMPO DETECCION BOMBA EN VACIO", in2 := 1000.0, out => #T4)
      { S7_Templates := "[SrcType := Real, DestType := DInt]" } Convert(in := #T4, out => #"Tiempo 4")
   END_RUNG
   RUNG wire#powerrail
      Mul(in1 := "CONFIG SIS AGUA POTABLE"."TIEMPO SLEEP BOOSTER", in2 := 1000.0, out => #T6)
      { S7_Templates := "[SrcType := Real, DestType := DInt]" } Convert(in := #T6, out => #"Tiempo 6")
   END_RUNG
   // the same network as SCL:
   #T1 := "CONFIG SIS AGUA POTABLE"."TIEMPO PARA MODO DORMIR" * 1000.0;
   #"Tiempo 1" := REAL_TO_DINT(#T1);
   #T2 := "CONFIG SIS AGUA POTABLE"."TIEMPO PARA ARRANCAR BOMBA EN PARALELO" * 1000.0;
   #"Tiempo 2" := REAL_TO_DINT(#T2);
   #T3 := "CONFIG SIS AGUA POTABLE"."TIEMPO PARA APAGAR BOMBA EN PARALELO" * 1000.0;
   #"Tiempo 3" := REAL_TO_DINT(#T3);
   #T4 := "CONFIG SIS AGUA POTABLE"."TIEMPO DETECCION BOMBA EN VACIO" * 1000.0;
   #"Tiempo 4" := REAL_TO_DINT(#T4);
   #T6 := "CONFIG SIS AGUA POTABLE"."TIEMPO SLEEP BOOSTER" * 1000.0;
   #"Tiempo 6" := REAL_TO_DINT(#T6);
END_REGION

REGION Network 2: FRECUENCIA DE OPERACION
   RUNG wire#powerrail
      Contact( "BOMBA LIDER 1" )
      Contact( "DISPONIBLE BOMBA A" )
      Move(in := "DATOS LECTURA VFDS"."096P004A".FRECUENCIA, out1 => #"FRECUENCIA OPERACION")
   END_RUNG
   RUNG wire#powerrail
      Contact( "BOMBA LIDER 2" )
      Contact( "DISPONIBLE BOMBA B" )
      Move(in := "DATOS LECTURA VFDS"."096P004B".FRECUENCIA, out1 => #"FRECUENCIA OPERACION")
   END_RUNG
   RUNG wire#powerrail
      Contact( "BOMBA LIDER 3" )
      Contact( "DISPONIBLE BOMBA C" )
      Move(in := "DATOS LECTURA VFDS"."096P004C".FRECUENCIA, out1 => #"FRECUENCIA OPERACION")
   END_RUNG
   RUNG wire#powerrail
      Contact( "BOMBA LIDER 4" )
      Contact( "DISPONIBLE BOMBA D" )
      Move(in := "DATOS LECTURA VFDS"."096P004D".FRECUENCIA, out1 => #"FRECUENCIA OPERACION")
   END_RUNG
   // the same network as SCL:
   IF "BOMBA LIDER 1" AND "DISPONIBLE BOMBA A" THEN
       #"FRECUENCIA OPERACION" := "DATOS LECTURA VFDS"."096P004A".FRECUENCIA;
   END_IF;
   IF "BOMBA LIDER 2" AND "DISPONIBLE BOMBA B" THEN
       #"FRECUENCIA OPERACION" := "DATOS LECTURA VFDS"."096P004B".FRECUENCIA;
   END_IF;
   IF "BOMBA LIDER 3" AND "DISPONIBLE BOMBA C" THEN
       #"FRECUENCIA OPERACION" := "DATOS LECTURA VFDS"."096P004C".FRECUENCIA;
   END_IF;
   IF "BOMBA LIDER 4" AND "DISPONIBLE BOMBA D" THEN
       #"FRECUENCIA OPERACION" := "DATOS LECTURA VFDS"."096P004D".FRECUENCIA;
   END_IF;
END_REGION

REGION Network 3: DORMIR DESPERTAR
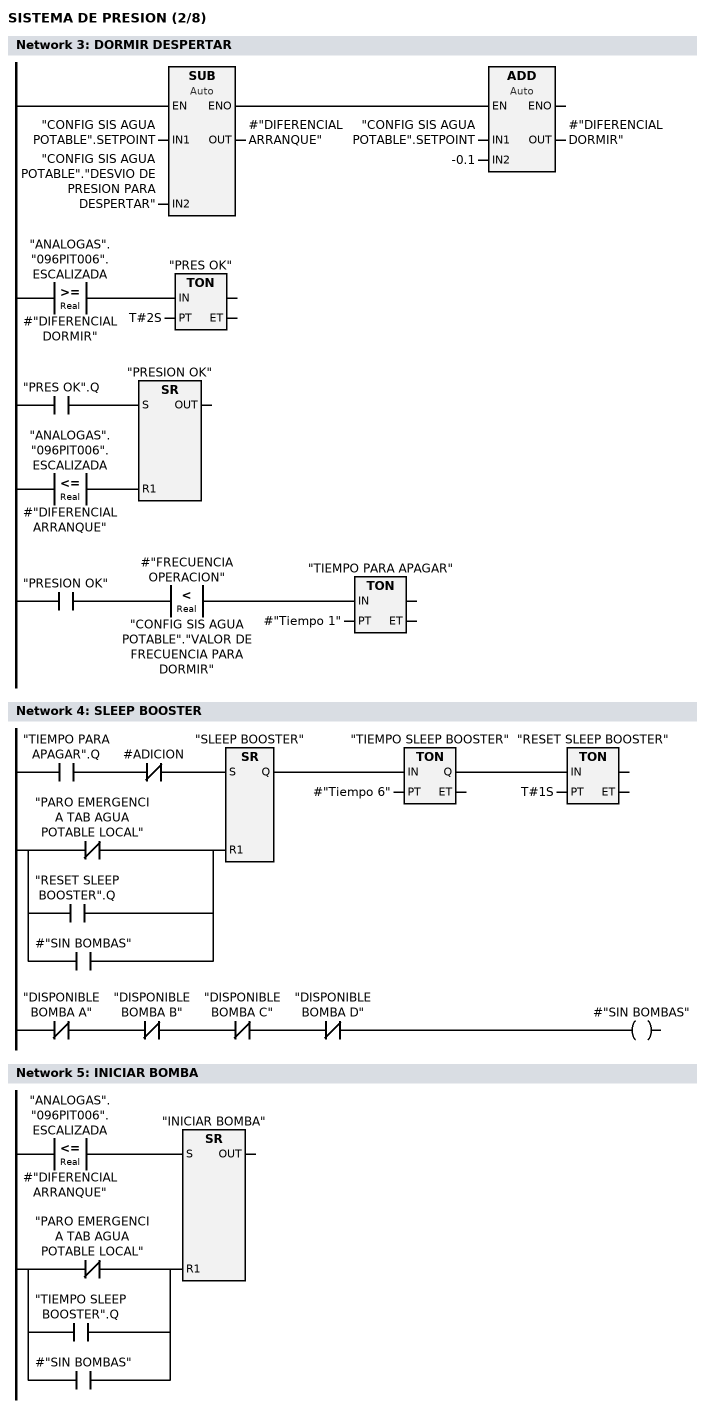
   #"DIFERENCIAL ARRANQUE" := "CONFIG SIS AGUA POTABLE".SETPOINT - "CONFIG SIS AGUA POTABLE"."DESVIO DE PRESION PARA DESPERTAR";
   #"DIFERENCIAL DORMIR" := "CONFIG SIS AGUA POTABLE".SETPOINT + (-0.1);
   "PRES OK".TON(IN := "ANALOGAS"."096PIT006".ESCALIZADA >= #"DIFERENCIAL DORMIR", PT := T#2S);
   IF "PRES OK".Q THEN
       "PRESION OK" := TRUE;   // SR flip-flop
   END_IF;
   IF "ANALOGAS"."096PIT006".ESCALIZADA <= #"DIFERENCIAL ARRANQUE" THEN "PRESION OK" := FALSE; END_IF;
   "TIEMPO PARA APAGAR".TON(IN := "PRESION OK" AND (#"FRECUENCIA OPERACION" < "CONFIG SIS AGUA POTABLE"."VALOR DE FRECUENCIA PARA DORMIR"),
                           PT := #"Tiempo 1");
END_REGION

REGION Network 4: SLEEP BOOSTER
   IF "TIEMPO PARA APAGAR".Q AND NOT #ADICION THEN
       "SLEEP BOOSTER" := TRUE;   // SR flip-flop
   END_IF;
   IF NOT "PARO EMERGENCIA TAB AGUA POTABLE LOCAL" OR "RESET SLEEP BOOSTER".Q OR #"SIN BOMBAS" THEN
       "SLEEP BOOSTER" := FALSE;
   END_IF;
   "TIEMPO SLEEP BOOSTER".TON(IN := "SLEEP BOOSTER", PT := #"Tiempo 6");
   "RESET SLEEP BOOSTER".TON(IN := "TIEMPO SLEEP BOOSTER".Q, PT := T#1S);
   #"SIN BOMBAS" := NOT "DISPONIBLE BOMBA A" AND NOT "DISPONIBLE BOMBA B" AND NOT "DISPONIBLE BOMBA C" AND NOT "DISPONIBLE BOMBA D";
END_REGION

REGION Network 5: INICIAR BOMBA
   RUNG wire#powerrail
      { S7_Templates := "SrcType := Real" } LE_Contact(in1 := "ANALOGAS"."096PIT006".ESCALIZADA, in2 := #"DIFERENCIAL ARRANQUE")
      S_SR(operand := "INICIAR BOMBA", r1 := wire#w1)
   END_RUNG
   RUNG wire#powerrail
      I_Contact( "PARO EMERGENCIA TAB AGUA POTABLE LOCAL" )
   END_RUNG wire#w1
   RUNG wire#powerrail
      Contact( "TIEMPO SLEEP BOOSTER".Q )
   END_RUNG wire#w1
   RUNG wire#powerrail
      Contact( #"SIN BOMBAS" )
   END_RUNG wire#w1
   // the same network as SCL:
   IF "ANALOGAS"."096PIT006".ESCALIZADA <= #"DIFERENCIAL ARRANQUE" THEN
       "INICIAR BOMBA" := TRUE;   // SR flip-flop
   END_IF;
   IF NOT "PARO EMERGENCIA TAB AGUA POTABLE LOCAL" OR "TIEMPO SLEEP BOOSTER".Q OR #"SIN BOMBAS" THEN
       "INICIAR BOMBA" := FALSE;
   END_IF;
END_REGION

REGION Network 6: CONTEO BOMBA A
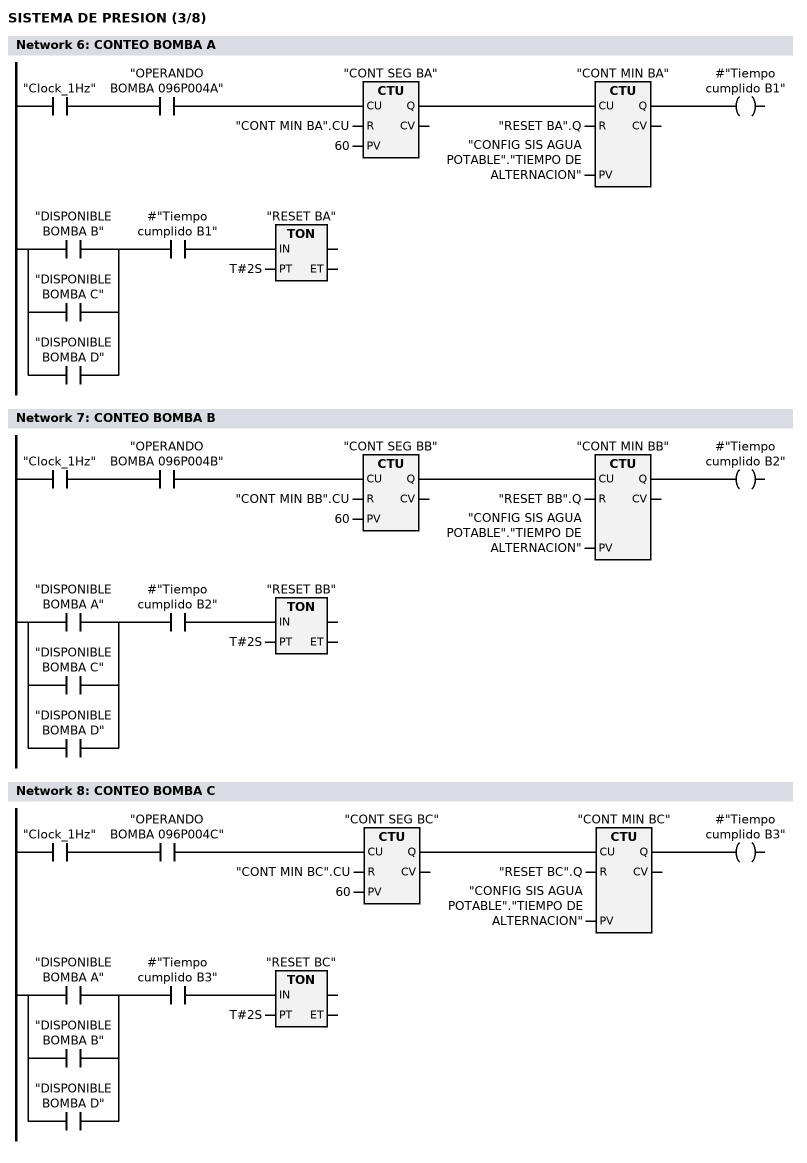
   "CONT SEG BA".CTU(CU := "Clock_1Hz" AND "OPERANDO BOMBA 096P004A", R := "CONT MIN BA".CU, PV := 60);
   "CONT MIN BA".CTU(CU := "CONT SEG BA".Q,
                     R := "RESET BA".Q,
                     PV := "CONFIG SIS AGUA POTABLE"."TIEMPO DE ALTERNACION");
   #"Tiempo cumplido B1" := "CONT MIN BA".Q;
   "RESET BA".TON(IN := ("DISPONIBLE BOMBA B" OR "DISPONIBLE BOMBA C" OR "DISPONIBLE BOMBA D") AND #"Tiempo cumplido B1",
                  PT := T#2S);
END_REGION

REGION Network 7: CONTEO BOMBA B
   "CONT SEG BB".CTU(CU := "Clock_1Hz" AND "OPERANDO BOMBA 096P004B", R := "CONT MIN BB".CU, PV := 60);
   "CONT MIN BB".CTU(CU := "CONT SEG BB".Q,
                     R := "RESET BB".Q,
                     PV := "CONFIG SIS AGUA POTABLE"."TIEMPO DE ALTERNACION");
   #"Tiempo cumplido B2" := "CONT MIN BB".Q;
   "RESET BB".TON(IN := ("DISPONIBLE BOMBA A" OR "DISPONIBLE BOMBA C" OR "DISPONIBLE BOMBA D") AND #"Tiempo cumplido B2",
                  PT := T#2S);
END_REGION

REGION Network 8: CONTEO BOMBA C
   "CONT SEG BC".CTU(CU := "Clock_1Hz" AND "OPERANDO BOMBA 096P004C", R := "CONT MIN BC".CU, PV := 60);
   "CONT MIN BC".CTU(CU := "CONT SEG BC".Q,
                     R := "RESET BC".Q,
                     PV := "CONFIG SIS AGUA POTABLE"."TIEMPO DE ALTERNACION");
   #"Tiempo cumplido B3" := "CONT MIN BC".Q;
   "RESET BC".TON(IN := ("DISPONIBLE BOMBA A" OR "DISPONIBLE BOMBA B" OR "DISPONIBLE BOMBA D") AND #"Tiempo cumplido B3",
                  PT := T#2S);
END_REGION

REGION Network 9: CONTEO BOMBA D
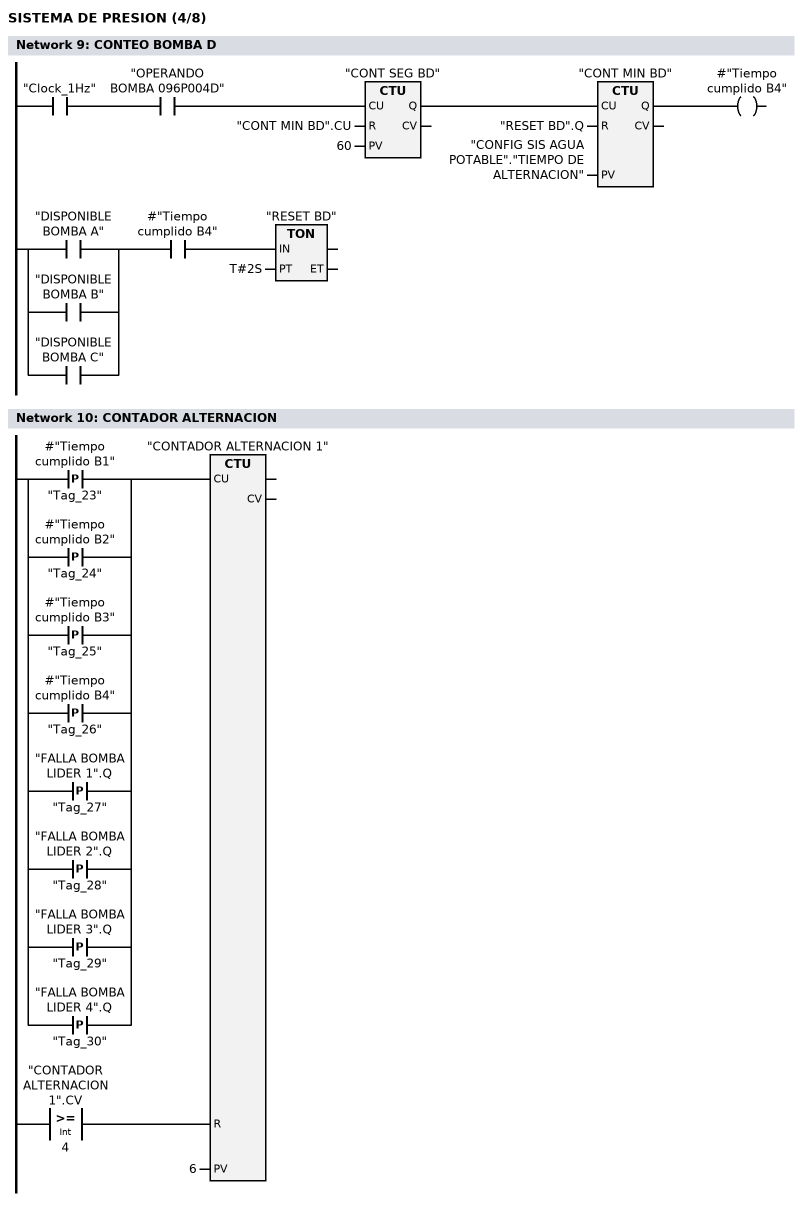
   "CONT SEG BD".CTU(CU := "Clock_1Hz" AND "OPERANDO BOMBA 096P004D", R := "CONT MIN BD".CU, PV := 60);
   "CONT MIN BD".CTU(CU := "CONT SEG BD".Q,
                     R := "RESET BD".Q,
                     PV := "CONFIG SIS AGUA POTABLE"."TIEMPO DE ALTERNACION");
   #"Tiempo cumplido B4" := "CONT MIN BD".Q;
   "RESET BD".TON(IN := ("DISPONIBLE BOMBA A" OR "DISPONIBLE BOMBA B" OR "DISPONIBLE BOMBA C") AND #"Tiempo cumplido B4",
                  PT := T#2S);
END_REGION

REGION Network 10: CONTADOR ALTERNACION
   #_w1 := #"Tiempo cumplido B1" AND NOT "Tag_23";   // rising edge of #"Tiempo cumplido B1"
   "Tag_23" := #"Tiempo cumplido B1";
   #_w2 := #"Tiempo cumplido B2" AND NOT "Tag_24";   // rising edge of #"Tiempo cumplido B2"
   "Tag_24" := #"Tiempo cumplido B2";
   #_w3 := #"Tiempo cumplido B3" AND NOT "Tag_25";   // rising edge of #"Tiempo cumplido B3"
   "Tag_25" := #"Tiempo cumplido B3";
   #_w4 := #"Tiempo cumplido B4" AND NOT "Tag_26";   // rising edge of #"Tiempo cumplido B4"
   "Tag_26" := #"Tiempo cumplido B4";
   #_w5 := "FALLA BOMBA LIDER 1".Q AND NOT "Tag_27";   // rising edge of "FALLA BOMBA LIDER 1".Q
   "Tag_27" := "FALLA BOMBA LIDER 1".Q;
   #_w6 := "FALLA BOMBA LIDER 2".Q AND NOT "Tag_28";   // rising edge of "FALLA BOMBA LIDER 2".Q
   "Tag_28" := "FALLA BOMBA LIDER 2".Q;
   #_w7 := "FALLA BOMBA LIDER 3".Q AND NOT "Tag_29";   // rising edge of "FALLA BOMBA LIDER 3".Q
   "Tag_29" := "FALLA BOMBA LIDER 3".Q;
   #_w8 := "FALLA BOMBA LIDER 4".Q AND NOT "Tag_30";   // rising edge of "FALLA BOMBA LIDER 4".Q
   "Tag_30" := "FALLA BOMBA LIDER 4".Q;
   "CONTADOR ALTERNACION 1".CTU(CU := #_w1 OR #_w2 OR #_w3 OR #_w4 OR #_w5 OR #_w6 OR #_w7 OR #_w8,
                           R := "CONTADOR ALTERNACION 1".CV >= 4,
                           PV := 6);
END_REGION

REGION Network 11: FALLA BOMBA LIDER
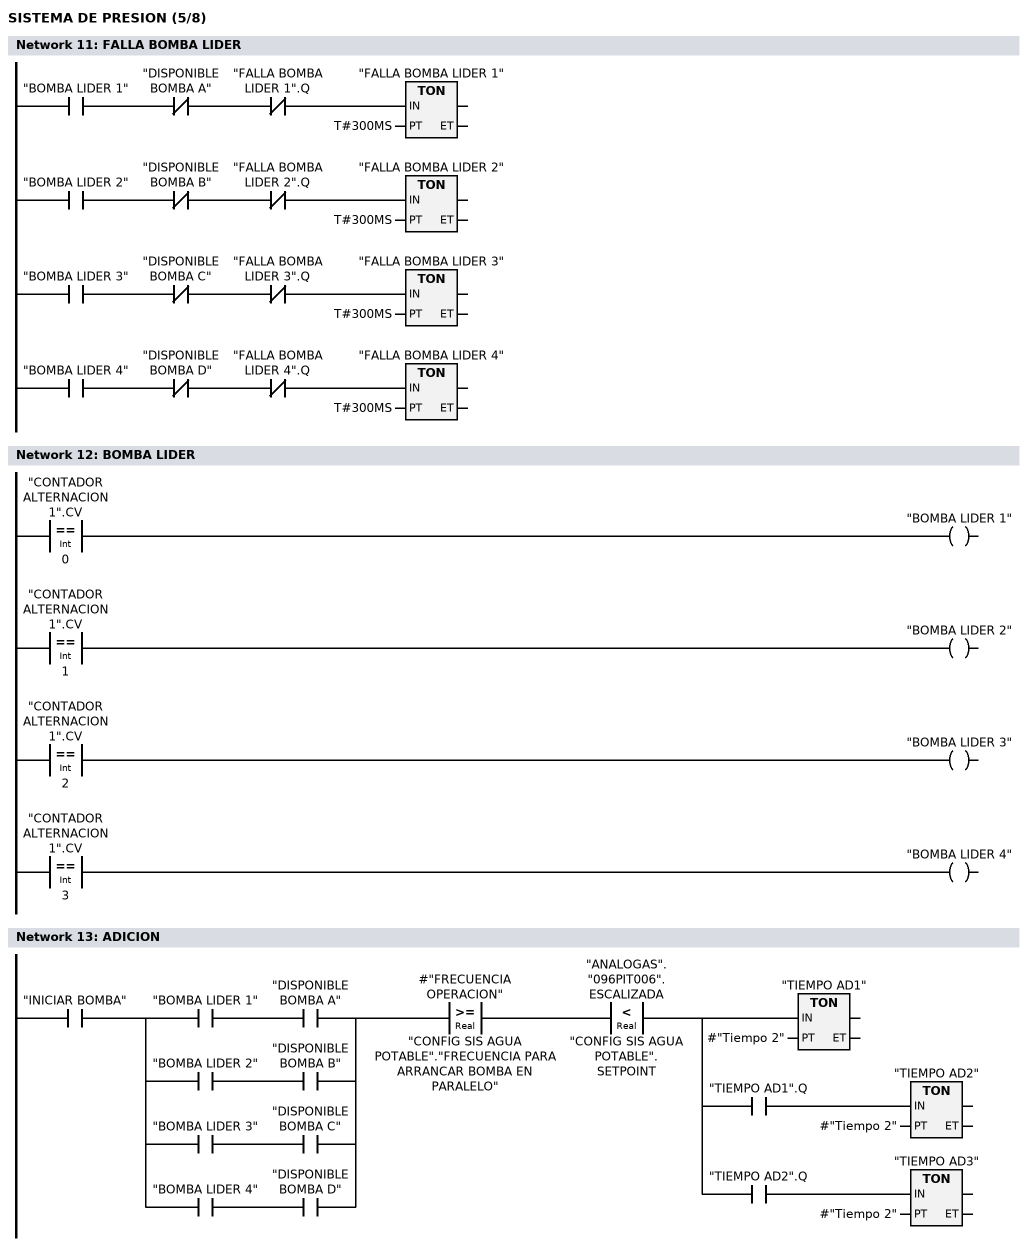
   "FALLA BOMBA LIDER 1".TON(IN := "BOMBA LIDER 1" AND NOT "DISPONIBLE BOMBA A" AND NOT "FALLA BOMBA LIDER 1".Q,
                           PT := T#300MS);
   "FALLA BOMBA LIDER 2".TON(IN := "BOMBA LIDER 2" AND NOT "DISPONIBLE BOMBA B" AND NOT "FALLA BOMBA LIDER 2".Q,
                           PT := T#300MS);
   "FALLA BOMBA LIDER 3".TON(IN := "BOMBA LIDER 3" AND NOT "DISPONIBLE BOMBA C" AND NOT "FALLA BOMBA LIDER 3".Q,
                           PT := T#300MS);
   "FALLA BOMBA LIDER 4".TON(IN := "BOMBA LIDER 4" AND NOT "DISPONIBLE BOMBA D" AND NOT "FALLA BOMBA LIDER 4".Q,
                           PT := T#300MS);
END_REGION

REGION Network 12: BOMBA LIDER
   RUNG wire#powerrail
      { S7_Templates := "SrcType := Int" } EQ_Contact(in1 := "CONTADOR ALTERNACION 1".CV, in2 := 0)
      Coil( "BOMBA LIDER 1" )
   END_RUNG
   RUNG wire#powerrail
      { S7_Templates := "SrcType := Int" } EQ_Contact(in1 := "CONTADOR ALTERNACION 1".CV, in2 := 1)
      Coil( "BOMBA LIDER 2" )
   END_RUNG
   RUNG wire#powerrail
      { S7_Templates := "SrcType := Int" } EQ_Contact(in1 := "CONTADOR ALTERNACION 1".CV, in2 := 2)
      Coil( "BOMBA LIDER 3" )
   END_RUNG
   RUNG wire#powerrail
      { S7_Templates := "SrcType := Int" } EQ_Contact(in1 := "CONTADOR ALTERNACION 1".CV, in2 := 3)
      Coil( "BOMBA LIDER 4" )
   END_RUNG
   // the same network as SCL:
   "BOMBA LIDER 1" := "CONTADOR ALTERNACION 1".CV = 0;
   "BOMBA LIDER 2" := "CONTADOR ALTERNACION 1".CV = 1;
   "BOMBA LIDER 3" := "CONTADOR ALTERNACION 1".CV = 2;
   "BOMBA LIDER 4" := "CONTADOR ALTERNACION 1".CV = 3;
END_REGION

REGION Network 13: ADICION
   #_w1 := "INICIAR BOMBA" AND (("BOMBA LIDER 1" AND "DISPONIBLE BOMBA A") OR ("BOMBA LIDER 2" AND "DISPONIBLE BOMBA B") OR ("BOMBA LIDER 3" AND "DISPONIBLE BOMBA C") OR ("BOMBA LIDER 4" AND "DISPONIBLE BOMBA D")) AND (#"FRECUENCIA OPERACION" >= "CONFIG SIS AGUA POTABLE"."FRECUENCIA PARA ARRANCAR BOMBA EN PARALELO") AND ("ANALOGAS"."096PIT006".ESCALIZADA < "CONFIG SIS AGUA POTABLE".SETPOINT);
   "TIEMPO AD1".TON(IN := #_w1, PT := #"Tiempo 2");
   "TIEMPO AD2".TON(IN := #_w1 AND "TIEMPO AD1".Q, PT := #"Tiempo 2");
   "TIEMPO AD3".TON(IN := #_w1 AND "TIEMPO AD2".Q, PT := #"Tiempo 2");
END_REGION

REGION Network 14: ADICION 1
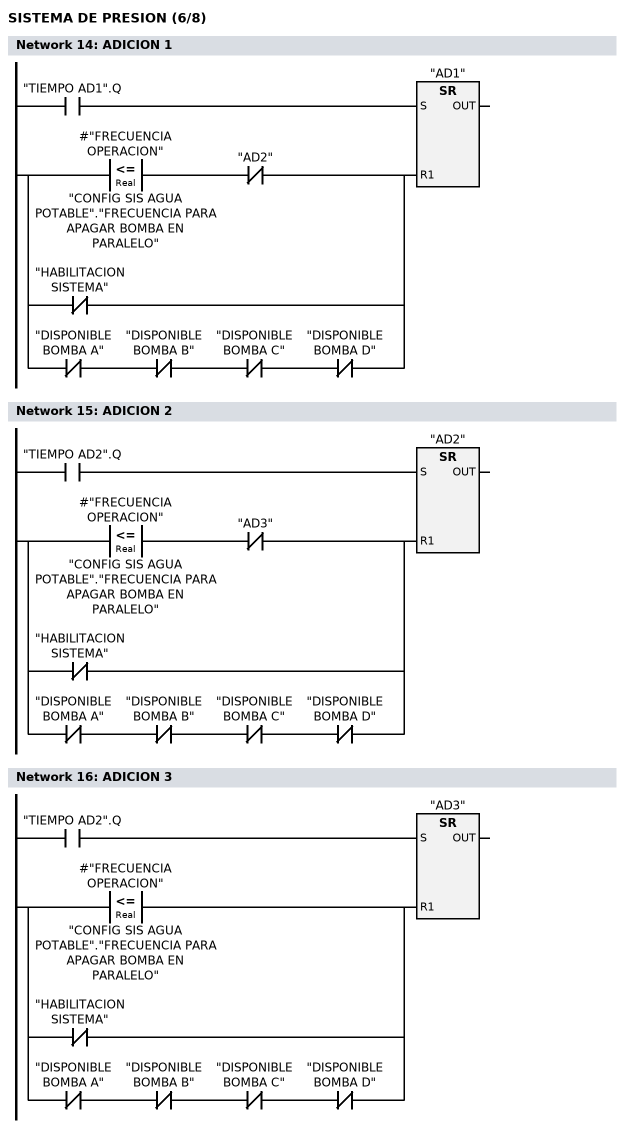
   RUNG wire#powerrail
      Contact( "TIEMPO AD1".Q )
      S_SR(operand := "AD1", r1 := wire#w1)
   END_RUNG
   RUNG wire#powerrail
      { S7_Templates := "SrcType := Real" } LE_Contact(in1 := #"FRECUENCIA OPERACION", in2 := "CONFIG SIS AGUA POTABLE"."FRECUENCIA PARA APAGAR BOMBA EN PARALELO")
      I_Contact( "AD2" )
   END_RUNG wire#w1
   RUNG wire#powerrail
      I_Contact( "HABILITACION SISTEMA" )
   END_RUNG wire#w1
   RUNG wire#powerrail
      I_Contact( "DISPONIBLE BOMBA A" )
      I_Contact( "DISPONIBLE BOMBA B" )
      I_Contact( "DISPONIBLE BOMBA C" )
      I_Contact( "DISPONIBLE BOMBA D" )
   END_RUNG wire#w1
   // the same network as SCL:
   IF "TIEMPO AD1".Q THEN
       "AD1" := TRUE;   // SR flip-flop
   END_IF;
   IF ((#"FRECUENCIA OPERACION" <= "CONFIG SIS AGUA POTABLE"."FRECUENCIA PARA APAGAR BOMBA EN PARALELO") AND NOT "AD2") OR NOT "HABILITACION SISTEMA" OR (NOT "DISPONIBLE BOMBA A" AND NOT "DISPONIBLE BOMBA B" AND NOT "DISPONIBLE BOMBA C" AND NOT "DISPONIBLE BOMBA D") THEN
       "AD1" := FALSE;
   END_IF;
END_REGION

REGION Network 15: ADICION 2
   RUNG wire#powerrail
      Contact( "TIEMPO AD2".Q )
      S_SR(operand := "AD2", r1 := wire#w1)
   END_RUNG
   RUNG wire#powerrail
      { S7_Templates := "SrcType := Real" } LE_Contact(in1 := #"FRECUENCIA OPERACION", in2 := "CONFIG SIS AGUA POTABLE"."FRECUENCIA PARA APAGAR BOMBA EN PARALELO")
      I_Contact( "AD3" )
   END_RUNG wire#w1
   RUNG wire#powerrail
      I_Contact( "HABILITACION SISTEMA" )
   END_RUNG wire#w1
   RUNG wire#powerrail
      I_Contact( "DISPONIBLE BOMBA A" )
      I_Contact( "DISPONIBLE BOMBA B" )
      I_Contact( "DISPONIBLE BOMBA C" )
      I_Contact( "DISPONIBLE BOMBA D" )
   END_RUNG wire#w1
   // the same network as SCL:
   IF "TIEMPO AD2".Q THEN
       "AD2" := TRUE;   // SR flip-flop
   END_IF;
   IF ((#"FRECUENCIA OPERACION" <= "CONFIG SIS AGUA POTABLE"."FRECUENCIA PARA APAGAR BOMBA EN PARALELO") AND NOT "AD3") OR NOT "HABILITACION SISTEMA" OR (NOT "DISPONIBLE BOMBA A" AND NOT "DISPONIBLE BOMBA B" AND NOT "DISPONIBLE BOMBA C" AND NOT "DISPONIBLE BOMBA D") THEN
       "AD2" := FALSE;
   END_IF;
END_REGION

REGION Network 16: ADICION 3
   RUNG wire#powerrail
      Contact( "TIEMPO AD2".Q )
      S_SR(operand := "AD3", r1 := wire#w1)
   END_RUNG
   RUNG wire#powerrail
      { S7_Templates := "SrcType := Real" } LE_Contact(in1 := #"FRECUENCIA OPERACION", in2 := "CONFIG SIS AGUA POTABLE"."FRECUENCIA PARA APAGAR BOMBA EN PARALELO")
   END_RUNG wire#w1
   RUNG wire#powerrail
      I_Contact( "HABILITACION SISTEMA" )
   END_RUNG wire#w1
   RUNG wire#powerrail
      I_Contact( "DISPONIBLE BOMBA A" )
      I_Contact( "DISPONIBLE BOMBA B" )
      I_Contact( "DISPONIBLE BOMBA C" )
      I_Contact( "DISPONIBLE BOMBA D" )
   END_RUNG wire#w1
   // the same network as SCL:
   IF "TIEMPO AD2".Q THEN
       "AD3" := TRUE;   // SR flip-flop
   END_IF;
   IF (#"FRECUENCIA OPERACION" <= "CONFIG SIS AGUA POTABLE"."FRECUENCIA PARA APAGAR BOMBA EN PARALELO") OR NOT "HABILITACION SISTEMA" OR (NOT "DISPONIBLE BOMBA A" AND NOT "DISPONIBLE BOMBA B" AND NOT "DISPONIBLE BOMBA C" AND NOT "DISPONIBLE BOMBA D") THEN
       "AD3" := FALSE;
   END_IF;
END_REGION

REGION Network 17: ARRANQUE B1
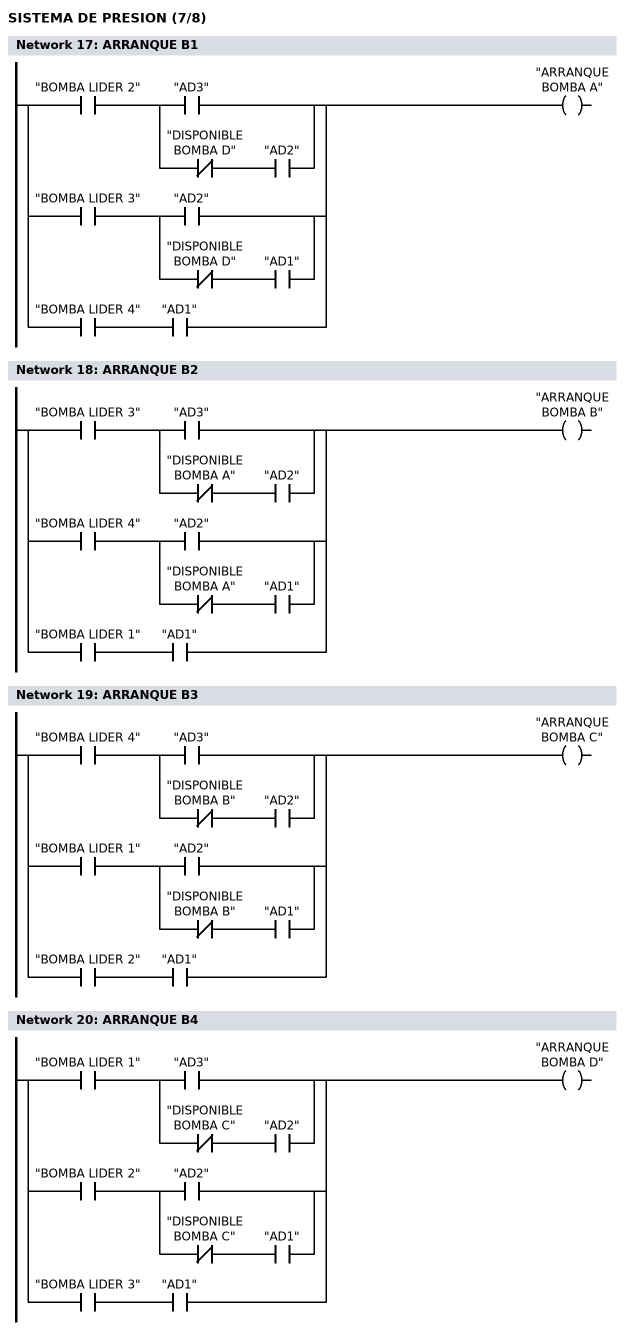
   RUNG wire#powerrail
      Contact( "BOMBA LIDER 2" )
      wire#w1
      Contact( "AD3" )
      wire#w2
      Coil( "ARRANQUE BOMBA A" )
   END_RUNG
   RUNG wire#w1
      I_Contact( "DISPONIBLE BOMBA D" )
      Contact( "AD2" )
   END_RUNG wire#w2
   RUNG wire#powerrail
      Contact( "BOMBA LIDER 3" )
      wire#w3
      Contact( "AD2" )
   END_RUNG wire#w2
   RUNG wire#w3
      I_Contact( "DISPONIBLE BOMBA D" )
      Contact( "AD1" )
   END_RUNG wire#w2
   RUNG wire#powerrail
      Contact( "BOMBA LIDER 4" )
      Contact( "AD1" )
   END_RUNG wire#w2
   // the same network as SCL:
   "ARRANQUE BOMBA A" := ("BOMBA LIDER 2" AND ("AD3" OR (NOT "DISPONIBLE BOMBA D" AND "AD2"))) OR ("BOMBA LIDER 3" AND ("AD2" OR (NOT "DISPONIBLE BOMBA D" AND "AD1"))) OR ("BOMBA LIDER 4" AND "AD1");
END_REGION

REGION Network 18: ARRANQUE B2
   RUNG wire#powerrail
      Contact( "BOMBA LIDER 3" )
      wire#w1
      Contact( "AD3" )
      wire#w2
      Coil( "ARRANQUE BOMBA B" )
   END_RUNG
   RUNG wire#w1
      I_Contact( "DISPONIBLE BOMBA A" )
      Contact( "AD2" )
   END_RUNG wire#w2
   RUNG wire#powerrail
      Contact( "BOMBA LIDER 4" )
      wire#w3
      Contact( "AD2" )
   END_RUNG wire#w2
   RUNG wire#w3
      I_Contact( "DISPONIBLE BOMBA A" )
      Contact( "AD1" )
   END_RUNG wire#w2
   RUNG wire#powerrail
      Contact( "BOMBA LIDER 1" )
      Contact( "AD1" )
   END_RUNG wire#w2
   // the same network as SCL:
   "ARRANQUE BOMBA B" := ("BOMBA LIDER 3" AND ("AD3" OR (NOT "DISPONIBLE BOMBA A" AND "AD2"))) OR ("BOMBA LIDER 4" AND ("AD2" OR (NOT "DISPONIBLE BOMBA A" AND "AD1"))) OR ("BOMBA LIDER 1" AND "AD1");
END_REGION

REGION Network 19: ARRANQUE B3
   RUNG wire#powerrail
      Contact( "BOMBA LIDER 4" )
      wire#w1
      Contact( "AD3" )
      wire#w2
      Coil( "ARRANQUE BOMBA C" )
   END_RUNG
   RUNG wire#w1
      I_Contact( "DISPONIBLE BOMBA B" )
      Contact( "AD2" )
   END_RUNG wire#w2
   RUNG wire#powerrail
      Contact( "BOMBA LIDER 1" )
      wire#w3
      Contact( "AD2" )
   END_RUNG wire#w2
   RUNG wire#w3
      I_Contact( "DISPONIBLE BOMBA B" )
      Contact( "AD1" )
   END_RUNG wire#w2
   RUNG wire#powerrail
      Contact( "BOMBA LIDER 2" )
      Contact( "AD1" )
   END_RUNG wire#w2
   // the same network as SCL:
   "ARRANQUE BOMBA C" := ("BOMBA LIDER 4" AND ("AD3" OR (NOT "DISPONIBLE BOMBA B" AND "AD2"))) OR ("BOMBA LIDER 1" AND ("AD2" OR (NOT "DISPONIBLE BOMBA B" AND "AD1"))) OR ("BOMBA LIDER 2" AND "AD1");
END_REGION

REGION Network 20: ARRANQUE B4
   RUNG wire#powerrail
      Contact( "BOMBA LIDER 1" )
      wire#w1
      Contact( "AD3" )
      wire#w2
      Coil( "ARRANQUE BOMBA D" )
   END_RUNG
   RUNG wire#w1
      I_Contact( "DISPONIBLE BOMBA C" )
      Contact( "AD2" )
   END_RUNG wire#w2
   RUNG wire#powerrail
      Contact( "BOMBA LIDER 2" )
      wire#w3
      Contact( "AD2" )
   END_RUNG wire#w2
   RUNG wire#w3
      I_Contact( "DISPONIBLE BOMBA C" )
      Contact( "AD1" )
   END_RUNG wire#w2
   RUNG wire#powerrail
      Contact( "BOMBA LIDER 3" )
      Contact( "AD1" )
   END_RUNG wire#w2
   // the same network as SCL:
   "ARRANQUE BOMBA D" := ("BOMBA LIDER 1" AND ("AD3" OR (NOT "DISPONIBLE BOMBA C" AND "AD2"))) OR ("BOMBA LIDER 2" AND ("AD2" OR (NOT "DISPONIBLE BOMBA C" AND "AD1"))) OR ("BOMBA LIDER 3" AND "AD1");
END_REGION

REGION Network 21: CONTADOR TRABAJO BOMBA A
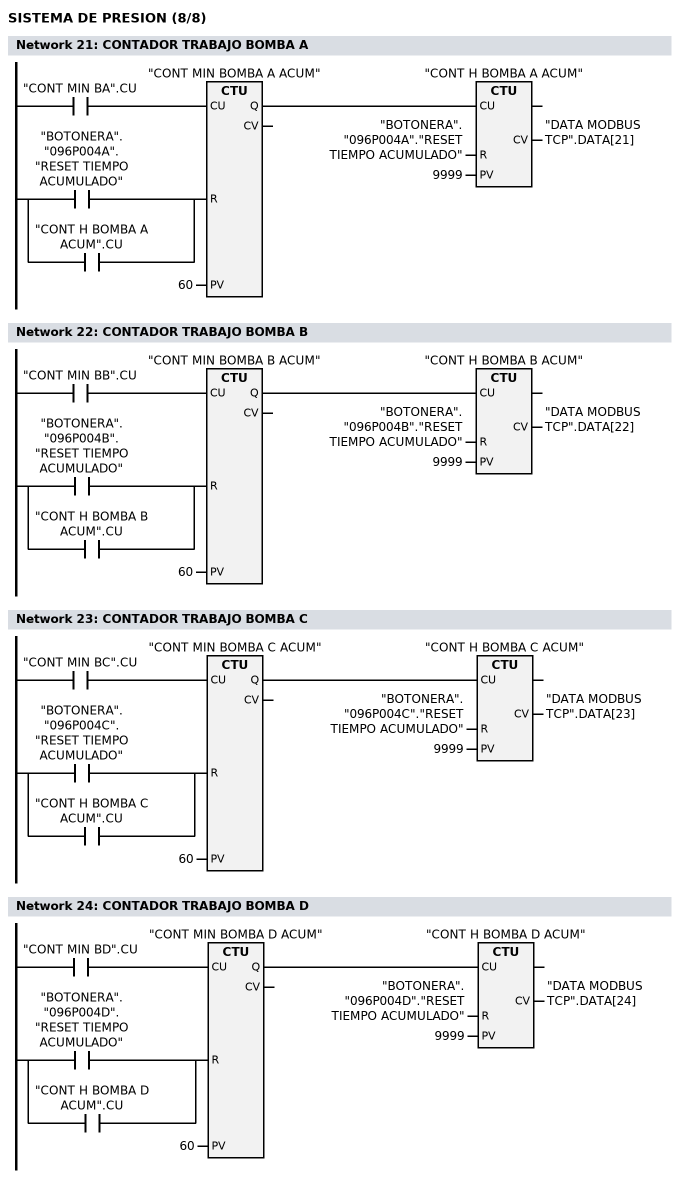
   "CONT MIN BOMBA A ACUM".CTU(CU := "CONT MIN BA".CU,
                           R := "BOTONERA"."096P004A"."RESET TIEMPO ACUMULADO" OR "CONT H BOMBA A ACUM".CU,
                           PV := 60);
   "CONT H BOMBA A ACUM".CTU(CU := "CONT MIN BOMBA A ACUM".Q,
                           R := "BOTONERA"."096P004A"."RESET TIEMPO ACUMULADO",
                           PV := 9999,
                           CV => "DATA MODBUS TCP".DATA[21]);
END_REGION

REGION Network 22: CONTADOR TRABAJO BOMBA B
   "CONT MIN BOMBA B ACUM".CTU(CU := "CONT MIN BB".CU,
                           R := "BOTONERA"."096P004B"."RESET TIEMPO ACUMULADO" OR "CONT H BOMBA B ACUM".CU,
                           PV := 60);
   "CONT H BOMBA B ACUM".CTU(CU := "CONT MIN BOMBA B ACUM".Q,
                           R := "BOTONERA"."096P004B"."RESET TIEMPO ACUMULADO",
                           PV := 9999,
                           CV => "DATA MODBUS TCP".DATA[22]);
END_REGION

REGION Network 23: CONTADOR TRABAJO BOMBA C
   "CONT MIN BOMBA C ACUM".CTU(CU := "CONT MIN BC".CU,
                           R := "BOTONERA"."096P004C"."RESET TIEMPO ACUMULADO" OR "CONT H BOMBA C ACUM".CU,
                           PV := 60);
   "CONT H BOMBA C ACUM".CTU(CU := "CONT MIN BOMBA C ACUM".Q,
                           R := "BOTONERA"."096P004C"."RESET TIEMPO ACUMULADO",
                           PV := 9999,
                           CV => "DATA MODBUS TCP".DATA[23]);
END_REGION

REGION Network 24: CONTADOR TRABAJO BOMBA D
   "CONT MIN BOMBA D ACUM".CTU(CU := "CONT MIN BD".CU,
                           R := "BOTONERA"."096P004D"."RESET TIEMPO ACUMULADO" OR "CONT H BOMBA D ACUM".CU,
                           PV := 60);
   "CONT H BOMBA D ACUM".CTU(CU := "CONT MIN BOMBA D ACUM".Q,
                           R := "BOTONERA"."096P004D"."RESET TIEMPO ACUMULADO",
                           PV := 9999,
                           CV => "DATA MODBUS TCP".DATA[24]);
END_REGION
END_FUNCTION

FUNCTION "COMUNICACION MODBUS TCP" : Void   // FC7, LAD
{ S7_Optimized_Access := 'TRUE' }
VERSION : 0.1
   VAR_TEMP
      "REAL 1" : Real;
      "REAL 2" : Real;
      "REAL 3" : Real;
      "REAL 4" : Real;
      "REAL 5" : Real;
      "REAL 6" : Real;
      "REAL 7" : Real;
      "REAL 8" : Real;
      "REAL 9" : Real;
      "REAL 10" : Real;
      "REAL 11" : Real;
      "REAL 12" : Real;
      "REAL 13" : Real;
      "REAL 14" : Real;
      "REAL 15" : Real;
      "REAL 16" : Real;
      "REAL 17" : Real;
      "REAL 18" : Real;
      "REAL 19" : Real;
      "REAL 20" : Real;
      "REAL 21" : Real;
      "REAL 22" : Real;
      "REAL 23" : Real;
      "REAL 24" : Real;
      "REAL 25" : Real;
      "REAL 26" : Real;
      "REAL 27" : Real;
      "REAL 28" : Real;
      "REAL 29" : Real;
      "REAL 30" : Real;
      T_CorrienteA : Real;
      T_CorrienteB : Real;
   END_VAR
   VAR_TEMP   // added for the SCL form of the ladder/FBD networks
      _w1 : Bool;
      _w2 : Bool;
      _w3 : Bool;
   END_VAR
BEGIN

REGION Network 1: CONFIGURACION MODBUS TCP
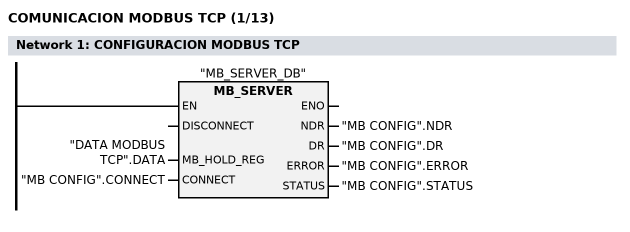
   "MB_SERVER_DB"(MB_HOLD_REG := "DATA MODBUS TCP".DATA,   // MB_SERVER
                  CONNECT := "MB CONFIG".CONNECT,
                  NDR => "MB CONFIG".NDR,
                  DR => "MB CONFIG".DR,
                  ERROR => "MB CONFIG".ERROR,
                  STATUS => "MB CONFIG".STATUS);
END_REGION

REGION Network 2: ENTRADAS DIGITALES
